Yaskawa INFORM job: OK_R2_O57-69(1)(90,0)_OK.JBI

/JOB
//NAME OK_R2_O57-69(1)(90,0)_OK
///FOLDERNAME X4
//POS
///NPOS 460,460,460,17,0,0
///TOOL 0
///POSTYPE PULSE
///PULSE
C00000=-107863,126513,61876,4074,92941,-4149
C00001=-107635,120046,52933,4022,95106,-4012
C00002=-107385,124787,62548,3925,91623,-4047
C00003=-107289,126429,66937,3891,89767,-4074
C00004=-107289,125685,67059,3890,89310,-4088
C00005=-107289,126429,66937,3891,89767,-4074
C00006=-107447,131976,74605,3936,87910,-4183
C00007=-107368,129085,70604,3913,88881,-4126
C00008=-107503,121805,59343,3962,92067,-4069
C00009=-107756,117289,50059,4061,95463,-4036
C00010=-108153,112100,52912,9904,92668,-10418
C00011=-107537,116907,62411,9707,89272,-10490
C00012=-107296,118643,67053,9639,87306,-10566
C00013=-107296,118210,67408,9641,86871,-10599
C00014=-107296,118643,67053,9639,87306,-10566
C00015=-106873,123308,73383,9530,85780,-10546
C00016=-107051,120523,69599,9574,86686,-10534
C00017=-107734,114067,59645,9761,89532,-10533
C00018=-108357,109439,50420,9963,92855,-10467
C00019=-111395,93808,29792,10909,97789,-10982
C00020=-122185,34205,35653,27729,49230,-19016
C00021=-120981,41909,45488,27980,46968,-19127
C00022=-117396,66636,64308,14609,59928,-14205
C00023=-117396,67398,66227,14722,59162,-14310
C00024=-117396,66924,65038,14651,59635,-14244
C00025=-117026,69424,68003,14605,59045,-14176
C00026=-117396,66924,65038,14651,59635,-14244
C00027=-121567,39659,44448,28509,46708,-19512
C00028=-122801,32028,34766,28268,48928,-19417
C00029=-122836,-30084,-33960,23424,71784,-41222
C00030=-108542,-18181,-29050,8736,76414,-35911
C00031=-108679,-18112,-25517,8852,74315,-36109
C00032=-108679,-17878,-23614,8896,73277,-36184
C00033=-108679,-18015,-24674,8871,73853,-36141
C00034=-101227,-12151,-22997,-5627,79968,-34149
C00035=-100809,-11793,-21323,-5732,79157,-33969
C00036=-99890,-11248,-20900,-5932,79243,-33658
C00037=-100809,-11793,-21323,-5732,79157,-33969
C00038=-119599,-28607,-38623,18108,79564,-38965
C00039=-143809,-13353,-27562,-4151,73883,-14363
C00040=-142866,3813,-3489,-4615,67955,-13814
C00041=-142866,4258,-993,-4658,66653,-13764
C00042=-142866,4067,-2013,-4640,67181,-13786
C00043=-143013,7668,1106,-4588,67106,-13835
C00044=-142866,4067,-2013,-4640,67181,-13786
C00045=-131729,19399,12333,-22118,77640,8494
C00046=-132684,19784,12695,-21959,77361,8191
C00047=-131729,18326,5882,-21907,80820,7904
C00048=-118180,-25123,-37779,-23861,88752,11312
C00049=-84402,-63677,-67114,-22586,99939,48241
C00050=-125926,-77250,-66316,-21080,81833,36437
C00051=-126284,-594,-20029,-15604,88354,35723
C00052=-126284,-509,-12976,-15645,84209,36248
C00053=-124802,3877,-7879,-15893,83645,36839
C00054=-124802,4020,-6552,-15911,82926,36931
C00055=-124802,3943,-7243,-15902,83298,36884
C00056=-123270,3785,-7378,-16131,83600,37383
C00057=-123399,3884,-6575,-16123,83149,37397
C00058=-123813,3922,-6544,-16060,83068,37263
C00059=-123399,3797,-7355,-16113,83568,37342
C00060=-129363,-46213,-49135,-15183,82438,35396
C00061=-131818,-93939,-91511,-4308,83147,7603
C00062=-129147,-104974,-80844,32439,31226,-48978
C00063=-125584,-72667,-62488,33742,33102,-67368
C00064=-122739,-67050,-57509,31022,31859,-65945
C00065=-121864,-64027,-53896,30654,30960,-65755
C00066=-121864,-63651,-52586,31182,30432,-66030
C00067=-121864,-64027,-53896,30654,30960,-65755
C00068=-121821,-59098,-51320,29827,31769,-65322
C00069=-121798,-56590,-49965,29444,32160,-65121
C00070=-121821,-59098,-51320,29827,31769,-65322
C00071=-130221,-55648,-47387,49393,39382,-72629
C00072=-128533,-55969,-47565,48393,38431,-72058
C00073=-122326,-63724,-54491,30711,31580,-65784
C00074=-123406,-65952,-56523,31749,32071,-66325
C00075=-126254,-71501,-61496,34397,33361,-67713
C00076=-120687,-90156,-48971,65843,10407,33929
C00077=-163424,-29173,-12092,69684,68620,47205
C00078=-167450,-15662,-2475,69350,71709,47134
C00079=-157670,-380,9649,68931,65290,48661
C00080=-176833,-62202,-56111,67907,81183,43629
C00081=-171503,-69579,-59831,67744,77015,43718
C00082=-167720,-72113,-59544,67781,73885,43604
C00083=-167720,-71727,-58313,67922,73661,43360
C00084=-167720,-72113,-59544,67781,73885,43604
C00085=-166558,-71597,-59299,67661,73156,43817
C00086=-165333,-70928,-58979,67520,72398,44056
C00087=-166558,-71597,-59299,67661,73156,43817
C00088=-171811,-70314,-60189,67797,77159,43607
C00089=-177694,-60868,-55413,67941,81861,43620
C00090=-178740,-64487,-57291,68086,82281,43176
C00091=-194893,-69888,-59984,68507,92693,40544
C00092=-214988,-85940,-67216,66402,104593,36100
C00093=-204042,-120915,-85873,62426,87530,23210
C00094=-200540,-66438,-67217,63628,100285,-15829
C00095=-127293,-88890,-117674,21964,112183,-47373
C00096=-127884,-113870,-117586,20406,100261,-49782
C00097=-126455,-94233,-83658,19548,96625,-49926
C00098=-122769,-95152,-80887,19686,93685,-49072
C00099=-121257,-92855,-76623,19731,91957,-48808
C00100=-121256,-92184,-75240,19721,91480,-48885
C00101=-121257,-92855,-76623,19731,91957,-48808
C00102=-119709,-92847,-76620,19813,91585,-48312
C00103=-118447,-92805,-76604,19874,91287,-47906
C00104=-121134,-93057,-78029,19757,92646,-48652
C00105=-122616,-92853,-79205,19699,93786,-49000
C00106=-126246,-91944,-81970,19569,96706,-49837
C00107=-116739,-91029,-87152,-11175,94833,69838
C00108=-118638,-93558,-84500,-11112,91693,69464
C00109=-121559,-94813,-81066,-11067,88585,68734
C00110=-121559,-94454,-79960,-11067,88097,68778
C00111=-121559,-94813,-81066,-11067,88585,68734
C00112=-121580,-97932,-82261,-11067,87731,68801
C00113=-121559,-94813,-81066,-11067,88585,68734
C00114=-124478,-94674,-81011,-11026,88221,67759
C00115=-121559,-94813,-81066,-11067,88585,68734
C00116=-121199,-93273,-83309,-11082,90766,68663
C00117=-119237,-90980,-86060,-11143,93854,69064
C00118=-119262,-91078,-98551,-11400,101347,68370
C00119=-119262,-88450,-105465,-11733,106843,67839
C00120=-123634,-129086,-124562,18007,62786,-21453
C00121=-124713,-112307,-109989,18584,62695,-21889
C00122=-121750,-102661,-104576,16897,63614,-20597
C00123=-120661,-96847,-100545,16291,63882,-20142
C00124=-120661,-96945,-99213,16408,63045,-20264
C00125=-120661,-96847,-100545,16291,63882,-20142
C00126=-119434,-96825,-100537,15680,63651,-19709
C00127=-118199,-96764,-100511,15059,63439,-19270
C00128=-119434,-96825,-100537,15680,63651,-19709
C00129=-120468,-95018,-99831,16130,64325,-20004
C00130=-120473,-92385,-98782,16042,65005,-19908
C00131=-120468,-95018,-99831,16130,64325,-20004
C00132=-121400,-102567,-103315,16828,62845,-20579
C00133=-124338,-112119,-108698,18515,61948,-21869
C00134=-115152,-110094,-108973,-21966,66789,27187
C00135=-118701,-101887,-103909,-20282,66922,25804
C00136=-120033,-96498,-99821,-19662,66842,25314
C00137=-120033,-96571,-98630,-19770,66116,25442
C00138=-120033,-96498,-99821,-19662,66842,25314
C00139=-121038,-96503,-99823,-19217,66607,24975
C00140=-122863,-96447,-99800,-18396,66209,24352
C00141=-121038,-96503,-99823,-19217,66607,24975
C00142=-121031,-93073,-98698,-19079,67622,24806
C00143=-121028,-91162,-97925,-19016,68103,24728
C00144=-121031,-93073,-98698,-19079,67622,24806
C00145=-119849,-101075,-102503,-19842,66224,25492
C00146=-116381,-109262,-107580,-21511,66068,26853
C00147=-114174,-113759,-109466,-25218,61256,29915
C00148=-117999,-105066,-104585,-23039,61495,28291
C00149=-119436,-99712,-100384,-22286,61259,27759
C00150=-119436,-99710,-99356,-22420,60673,27881
C00151=-119436,-99712,-100384,-22286,61259,27759
C00152=-121229,-99730,-100389,-21374,60785,27131
C00153=-123455,-99637,-100354,-20211,60254,26337
C00154=-121229,-99730,-100389,-21374,60785,27131
C00155=-121193,-87849,-97584,-20616,64895,26352
C00156=-121184,-85182,-96456,-20515,65531,26236
C00157=-121193,-87849,-97584,-20616,64895,26352
C00158=-119818,-94456,-100985,-21520,64018,27049
C00159=-116346,-102514,-105912,-23431,63914,28430
C00160=-120616,-96535,-104175,-23887,64719,45568
C00161=-120616,-96992,-102054,-24182,63306,45881
C00162=-136549,-91664,-102215,-2850,64532,40154
C00163=-118869,-97062,-101163,-25162,63282,46587
C00164=-120614,-98220,-102778,-24220,63138,45920
C00165=-133771,-94843,-111628,-11760,91195,37379
C00166=-135495,-95953,-105009,-10406,87462,38794
C00167=-135817,-95923,-103691,-10152,86855,39072
C00168=-120616,-96793,-103087,-23408,87451,42960
C00169=-120617,-96070,-105685,-23410,89266,42604
C00170=-120635,-118119,-124325,-17957,114364,37370
C00171=-107148,-122068,-106720,-37591,45003,56343
C00172=-107143,-118125,-97071,-40168,41922,57944
C00173=-107140,-117153,-94914,-40772,41285,58308
C00174=-108761,-111076,-92035,-38763,41593,57087
C00175=-105115,-116142,-93852,-42098,42144,59139
C00176=-107012,-118507,-95796,-40965,41228,58425
C00177=-106625,-124982,-112623,-27698,77800,49761
C00178=-108670,-124346,-112001,-25564,83023,48254
C00179=-122914,-112386,-108022,-9565,118901,48106
C00180=-107149,-124464,-114807,-14035,115464,42498
C00181=-107153,-124980,-118069,-14274,117155,42276
C00182=-120683,-72727,-118704,-1403,106780,1205
C00183=-120616,-97084,-101761,23685,56760,-46645
C00184=-120615,-97341,-97713,24403,54354,-47226
C00185=-120615,-97245,-95574,24781,53197,-47519
C00186=-113473,-96585,-93861,15515,48754,-41599
C00187=-120613,-98403,-96349,24817,53089,-47545
C00188=-122362,-97151,-94697,25998,53280,-48291
C00189=-118726,-95773,-106258,22948,89010,-41713
C00190=-118527,-107245,-109313,22939,85243,-42364
C00191=-120617,-95328,-107797,23350,90604,-42068
C00192=-120618,-93989,-110172,23402,92584,-41681
C00193=-120619,-87370,-116055,23793,99045,-40394
C00194=-120619,-87370,-116055,23793,99045,-40394
C00195=-120618,-86394,-114990,-8935,74593,-77376
C00196=-120618,-89943,-112390,-9089,71210,-77123
C00197=-120618,-91094,-111253,-9157,69935,-77026
C00198=-120921,-87010,-110025,-8929,71231,-77225
C00199=-120616,-91696,-112687,-9127,70502,-77069
C00200=-120617,-91433,-110915,-9280,69085,-76949
C00201=-120617,-91707,-110620,-9342,68290,-76888
C00202=-120617,-92092,-110153,-9289,66860,-76810
C00203=-120617,-92703,-109346,-8604,64312,-76688
C00204=-120617,-93084,-108807,-7222,62458,-76641
C00205=-120617,-93193,-108666,-5837,61715,-76664
C00206=-120618,-90875,-111661,-5103,64613,-76670
C00207=-120618,-90809,-111742,-4197,64653,-76687
C00208=-120618,-90545,-112027,-2634,65244,-76730
C00209=-120618,-90001,-112556,-1051,66686,-76779
C00210=-120618,-89211,-113241,130,68806,-76818
C00211=-120618,-88484,-113805,667,70701,-76840
C00212=-120618,-87123,-114601,725,72803,-76709
C00213=-120619,-86169,-115177,666,75079,-76754
C00214=-120619,-85009,-115798,-44,77805,-76866
C00215=-120619,-84186,-116189,-1368,79788,-77043
C00216=-120619,-83945,-116287,-2643,80551,-77203
C00217=-118270,-87908,-113898,-4548,77310,-76315
C00218=-117006,-87882,-113777,-5977,77383,-75992
C00219=-115001,-87936,-113393,-8376,77055,-75464
C00220=-113157,-88199,-112730,-10795,75966,-74930
C00221=-112003,-88721,-111920,-12625,74164,-74513
C00222=-111959,-89151,-111512,-13141,72976,-74431
C00223=-114352,-90005,-111461,-12180,71784,-75105
C00224=-117604,-90791,-111341,-10710,70486,-76060
C00225=-117404,-89600,-112462,-10735,71791,-76111
C00226=-116906,-85938,-115017,-10812,75246,-76259
C00227=-120614,-97623,-100799,-20300,88883,51757
C00228=-120614,-96302,-87355,-20440,81742,52958
C00229=-120613,-95405,-83784,-20521,80111,53236
C00230=-127344,-108772,-84900,-17713,65232,40253
C00231=-119108,-93712,-82042,-20736,80300,53753
C00232=-120703,-96440,-84059,-20528,79748,53266
C00233=-121654,-94959,-82200,-16195,85067,56749
C00234=-121447,-94482,-79045,-16244,83477,57034
C00235=-120534,-97306,-80078,-13287,88870,68293
C00236=-120613,-95181,-82964,-13310,91650,67966
C00237=-120614,-96223,-86939,-13345,93512,67766
C00238=-120615,-97634,-95801,-13498,98116,67263
C00239=-121294,-114205,-91205,24827,58618,-34956
C00240=-120612,-94063,-79189,30374,49118,-27390
C00241=-120612,-92317,-74276,31337,47279,-28045
C00242=-120611,-91635,-72532,31685,46659,-28276
C00243=-117825,-85297,-69483,27706,45876,-25590
C00244=-120609,-92794,-73597,31655,46709,-28256
C00245=-122365,-91337,-71823,32796,47086,-29053
C00246=-115287,-110447,-90354,20374,67075,-37718
C00247=-116232,-100454,-77072,21254,66209,-40580
C00248=-116013,-94136,-76050,20295,81458,-56297
C00249=-120612,-93792,-78416,23522,88402,-60481
C00250=-120613,-94966,-82014,23532,89885,-60189
C00251=-192979,-49879,-84133,31949,90821,-59300
C00252=-226136,-49296,-77583,43048,96139,-60221
C00253=-194231,-43574,-37464,64429,96533,35524
C00254=-168190,-921,2356,69742,86936,65420
C00255=-167171,-9679,-4727,69794,80481,66551
C00256=-161668,-12899,-4972,71887,72051,48991
C00257=-157343,-12771,-6150,68681,68498,39910
C00258=-156881,-17849,-10944,69825,79076,66625
C00259=-156054,-17027,-11609,69675,78824,67093
C00260=-157320,-12846,-6207,68680,68481,39912
C00261=-155303,-14498,-7398,68413,65801,40416
C00262=-150761,-18705,-10675,67104,57790,42164
C00263=-154138,4950,8277,69166,76187,38481
C00264=-154445,-11009,-7055,66235,75211,55885
C00265=-154064,-10379,-10377,61252,81435,65690
C00266=-159305,-13086,-7363,68622,70046,39902
C00267=-160610,-11568,-6196,68690,70948,39749
C00268=-179726,-19719,-12316,69264,83687,37039
C00269=-180202,-65513,-36112,70171,79517,38597
C00270=-171321,-47804,-23743,70196,73038,45095
C00271=-120855,-117042,-83065,287,50429,-281
C00272=-120852,-56541,-79529,233,79340,-219
C00273=-120696,51333,26745,175,69370,-180
C00274=-120686,107911,74673,172,68949,-177
C00275=-120685,95088,60632,169,71000,-174
C00276=-122318,97205,64688,817,69601,-751
C00277=-120685,108202,77433,173,67399,-179
C00278=-120704,104217,73450,180,67803,-185
C00279=-122286,97202,64700,804,69591,-740
C00280=-121454,98107,65862,475,69334,-448
C00281=-120585,97922,65623,2034,69446,-1841
C00282=-122017,99369,67601,7878,69886,-7136
C00283=-124401,105713,75936,15606,71119,-14640
C00284=-128119,115493,91326,26372,70058,-18277
C00285=-128088,115464,91288,26362,70055,-18265
C00286=-119886,111402,95174,38234,57086,-30403
C00287=-120666,108818,81293,29360,75518,-26461
C00288=-140740,108253,75800,14319,69459,-12393
C00289=-141155,96820,62941,14306,71509,-12294
C00290=-143909,115216,86261,19079,74712,-18279
C00291=-140740,108512,78347,14450,68068,-12565
C00292=-141173,105757,75971,14609,68190,-12710
C00293=-142377,104065,71962,18453,77277,-17320
C00294=-143915,117471,89727,22794,77825,-23537
C00295=-139477,109798,84410,35996,86879,-36501
C00296=-140751,108928,81956,36051,87607,-36108
C00297=-140752,108346,78971,36051,88864,-35697
C00298=-147823,62894,38016,27898,90947,-27507
C00299=-160213,20954,5847,52912,104038,-48859
C00300=-159152,20729,17995,59071,100827,-50067
C00301=-155802,40777,37843,59069,97737,-50212
C00302=-160195,38796,31307,59203,102054,-49818
C00303=-156773,55935,3033,15469,106475,-467
C00304=-153918,39963,-12238,-14336,97152,19223
C00305=-159942,42906,-84,-7000,88493,12017
C00306=-161832,44450,4966,-4658,85344,9495
C00307=-160451,43537,6688,-5079,83896,9996
C00308=-170176,47751,11203,12092,85800,-8664
C00309=-172574,61876,26837,20283,90605,-20342
C00310=-175474,59660,23243,20803,92313,-21058
C00311=-176824,52719,4578,21456,100048,-20156
C00312=-152577,48148,-11201,-5231,110173,9097
C00313=-182779,-40861,-76585,4205,87735,83212
C00314=-189334,-126614,-108463,44477,62316,64668
C00315=-120096,-126434,-88762,51835,16555,74218
C00316=-139248,-82584,-73342,59042,45862,69599
C00317=-136350,-83647,-73803,58003,43942,70198
C00318=-130421,-76673,-73912,46604,46265,76427
C00319=-135820,-86240,-74234,58721,43036,69743
C00320=-135177,-84196,-74622,57263,43352,70634
C00321=-130462,-76664,-73908,46626,46288,76415
C00322=-118284,-90424,-77484,27464,26422,76602
C00323=-134750,-71454,-68054,46452,38063,58888
C00324=-143711,-58767,-60463,57749,51756,38253
C00325=-120675,-86248,-74914,23863,24288,53303
C00326=-120674,-86256,-74917,23863,24286,53303
C00327=-120096,-126434,-88762,51835,16555,74218
C00328=-118534,-85327,-101542,-31688,82312,3081
C00329=-123235,4833,-40404,-29868,88268,-211
C00330=-160796,40344,30640,-17217,54638,-7315
C00331=-160797,40341,30637,-17217,54638,-7315
C00332=-160797,40341,30637,-17217,54638,-7315
C00333=-160252,39151,28676,-17378,55324,-7200
C00334=-161178,38223,28434,-16963,54814,-7508
C00335=-160796,40350,30646,-17218,54637,-7315
C00336=-160795,40351,30648,-17218,54637,-7314
C00337=-160794,40354,30651,-17218,54637,-7314
C00338=-134054,6396,-12292,-27269,70214,305
C00339=-134055,6392,-12295,-27269,70214,305
C00340=-134055,6392,-12295,-27269,70214,305
C00341=-133335,6117,-13247,-27465,70843,432
C00342=-134208,4264,-14132,-27207,70198,248
C00343=-134055,6400,-12288,-27269,70214,305
C00344=-134054,6402,-12286,-27269,70214,305
C00345=-134054,6405,-12283,-27270,70214,305
C00346=-134054,6378,-12307,-27269,70215,305
C00347=-110297,97127,46558,-158,86609,-5885
C00348=-106536,103923,39499,6534,95353,-6477
C00349=-105914,112602,52325,6316,91893,-6465
C00350=-107411,115180,62232,6738,87264,-7175
C00351=-107307,119116,66280,6709,86790,-7167
C00352=-105927,112591,52310,6320,91897,-6469
C00353=-107439,122836,73336,-765,83341,-3278
C00354=-107821,123137,73841,-645,83181,-3398
C00355=-102914,145277,103073,-11065,82212,10729
C00356=-102506,149279,108574,-13236,82700,14235
C00357=-102941,142782,99507,-15695,87156,18184
C00358=-102438,125149,73506,-15865,93942,17486
C00359=-103348,95167,36366,-12069,90690,17205
C00360=-107306,118463,66661,-801,85196,-3245
C00361=-107311,128667,66498,14067,94509,-10827
C00362=-105409,128969,69208,9127,93984,-11176
C00363=-104752,117595,57274,7632,88999,-11570
C00364=-107310,126688,66629,14039,93443,-10948
C00365=-107566,122823,62593,14116,93966,-10970
C00366=-105955,108102,46748,11418,87672,-11524
C00367=-106075,110081,48628,12407,89224,-11272
C00368=-104774,107445,45071,11972,89867,-10810
C00369=-104167,107349,44943,11766,89817,-10628
C00370=-103614,108174,46048,11576,89495,-10489
C00371=-105019,105279,39955,12261,92654,-10576
C00372=-107312,128730,66586,14067,94488,-10830
C00373=-113054,107191,42951,15619,98894,-12042
C00374=-132655,20555,-34602,20500,105579,-17250
C00375=-120395,-75677,-109491,17431,99945,-14261
C00376=-120731,-81008,-115648,-105,86416,-81801
C00377=-120675,-24654,-47163,-132,73228,-81771
C00378=-120676,-24640,-47153,-131,73229,-81771
C00379=-121102,-22780,-44290,48,72423,-81914
C00380=-120676,-24370,-48215,-131,74021,-81772
C00381=-121750,-24626,-47144,317,73232,-82133
C00382=-121088,-18910,-41523,41,72708,-81911
C00383=-120676,-24640,-47153,-131,73229,-81771
C00384=-120672,-32524,-49889,-133,70864,-81769
C00385=-86683,-40445,-63075,-13763,77736,-70672
C00386=-103499,26970,-9106,-7161,77072,-76192
C00387=-140778,108078,66600,-20509,92089,-48724
C00388=-140778,108101,66629,-20508,92083,-48723
C00389=-140777,108123,66659,-20508,92077,-48722
C00390=-140791,110557,71328,-20474,90549,-48468
C00391=-140777,108420,65802,-20527,92715,-48830
C00392=-141368,109052,67884,-20414,91674,-48860
C00393=-140538,117676,80864,-20492,88534,-48038
C00394=-140777,108123,66659,-20508,92077,-48722
C00395=-140778,108101,66629,-20508,92083,-48723
C00396=-140778,108101,66629,-20508,92083,-48723
C00397=-140778,108122,66658,-20508,92077,-48722
C00398=-140768,108703,68758,-20489,91145,-48562
C00399=-140777,108420,65801,-20527,92715,-48830
C00400=-141368,109051,67883,-20414,91674,-48860
C00401=-140511,115176,77354,-20500,89363,-48171
C00402=-140778,108122,66658,-20508,92077,-48722
C00403=-140778,108100,66628,-20508,92083,-48723
C00404=-140778,108078,66599,-20509,92089,-48724
C00405=-126581,14025,-47477,-25241,115824,-48542
C00406=-159492,92702,46653,-29136,105568,-44545
C00407=-162149,88036,41181,-28914,105145,-45798
C00408=-163325,88052,47564,-28312,101300,-45262
C00409=-160866,111719,71725,-28335,100123,-43674
C00410=-160864,108336,66000,-28535,101703,-44070
C00411=-164354,88224,47874,-28236,100875,-45547
C00412=-160866,108108,66623,-28476,101259,-43959
C00413=-161429,110004,69125,-28389,100573,-44000
C00414=-160867,107600,68720,-43807,97992,-44930
C00415=-160869,107245,72152,-43546,96305,-44200
C00416=-160853,112270,81548,-43267,93953,-43186
C00417=-160872,111361,79145,-43345,94689,-43509
C00418=-160869,107230,72446,-43527,96165,-44140
C00419=-161852,112523,81931,-43214,93388,-43402
C00420=-160870,107231,72133,-43547,96307,-44201
C00421=-160868,107586,68702,-43807,97995,-44932
C00422=-160873,107541,68625,-43810,98010,-44941
C00423=-160875,107181,72050,-43549,96324,-44211
C00424=-160969,112164,81513,-43259,93871,-43205
C00425=-160878,111286,79028,-43348,94711,-43521
C00426=-160875,107165,72344,-43530,96184,-44151
C00427=-161946,112277,81723,-43208,93342,-43426
C00428=-160876,107167,72031,-43549,96326,-44212
C00429=-160874,107528,68607,-43810,98012,-44942
C00430=-160865,108116,66633,-19225,80466,79641
C00431=-160864,108012,67019,-19239,80191,79685
C00432=-160902,111102,73963,-19378,77641,80084
C00433=-160868,111461,73140,-19346,78303,79987
C00434=-160865,107941,67240,-19247,80028,79711
C00435=-161896,111383,74336,-19093,77331,79779
C00436=-160866,107998,67001,-19238,80195,79684
C00437=-160866,108102,66615,-19224,80470,79640
C00438=-141960,25007,-13534,-18907,77065,75548
C00439=-148396,38776,-224,-4331,80270,75408
C00440=-147937,42862,4060,-4507,79758,75574
C00441=-147586,38479,-2882,-4613,81790,75612
C00442=-132676,28155,-16568,-22865,92034,69453
C00443=-139622,-24488,-52979,-20482,85647,66084
C00444=-105595,-117820,-100492,-25848,75539,72989
C00445=-106580,-108863,-97500,-25415,77736,72126
C00446=-109054,-118504,-91401,-16987,64899,66879
C00447=-114351,-116427,-87550,-15194,62531,65147
C00448=-119485,-94955,-76898,-12502,65960,62737
C00449=-99170,-109633,-81201,-29999,68590,70531
C00450=-97263,-108225,-79726,-30318,69111,71170
C00451=-119688,-71486,-66798,-11989,71648,62069
C00452=-119489,-72073,-70371,-11931,73536,61952
C00453=-119715,-43131,-54580,-11630,78554,61387
C00454=-119934,-43288,-51446,-11646,76556,61502
C00455=-120006,-17553,-34071,-11532,79027,61243
C00456=-119832,-16968,-37707,-11506,81540,61066
C00457=-138269,-21321,-44343,15851,46320,74175
C00458=-176671,-154466,-104215,64912,39697,45563
C00459=-34524,-124554,-102946,40349,70974,61921
BC00000=290556,778984,53
BC00001=296477,827832,53
BC00002=296477,827832,53
BC00003=296477,827832,52
BC00004=296477,827832,52
BC00005=296477,827832,52
BC00006=296477,827832,52
BC00007=296477,827832,52
BC00008=296477,827832,53
BC00009=296477,827832,53
BC00010=305680,824697,66927
BC00011=305680,824697,66927
BC00012=305680,824697,66927
BC00013=305680,824697,66927
BC00014=305680,824697,66927
BC00015=305680,824697,66927
BC00016=305680,824697,66927
BC00017=305680,824697,66927
BC00018=305680,824697,66927
BC00019=305680,824697,66927
BC00020=269068,808420,256770
BC00021=269068,808420,256770
BC00022=269068,808420,256770
BC00023=269068,808420,256770
BC00024=269068,808420,256770
BC00025=269068,808420,256770
BC00026=269068,808420,256770
BC00027=269068,808420,256770
BC00028=269068,808420,256770
BC00029=269068,808420,256770
BC00030=269068,808420,256770
BC00031=269068,808420,256770
BC00032=269068,808420,256770
BC00033=269068,808420,256770
BC00034=269068,808420,256770
BC00035=269068,808420,256770
BC00036=269068,808420,256770
BC00037=269068,808420,256770
BC00038=269068,808420,256770
BC00039=269068,808420,256770
BC00040=269068,808420,256770
BC00041=269068,808420,256770
BC00042=269068,808420,256770
BC00043=269068,808420,256770
BC00044=269068,808420,256770
BC00045=269068,808420,256770
BC00046=269068,808420,256770
BC00047=269068,808420,256770
BC00048=269068,808420,256770
BC00049=269068,722620,256770
BC00050=178494,722620,256770
BC00051=178494,722620,256770
BC00052=178494,722620,256770
BC00053=178494,722620,256770
BC00054=178494,722620,256770
BC00055=178494,722620,256770
BC00056=178494,722620,256770
BC00057=178494,722620,256770
BC00058=178494,722620,256770
BC00059=178494,722620,256770
BC00060=178494,722620,256770
BC00061=138756,709064,202273
BC00062=61964,682869,96959
BC00063=15,683519,90542
BC00064=15,683519,90542
BC00065=15,683519,90542
BC00066=15,683519,90542
BC00067=15,683519,90542
BC00068=15,683519,90542
BC00069=15,683519,90542
BC00070=15,683519,90542
BC00071=15,683519,90542
BC00072=15,683519,90542
BC00073=15,683519,90542
BC00074=15,683519,90542
BC00075=15,683519,90542
BC00076=1273,683756,232707
BC00077=15,671225,229408
BC00078=15,671225,229408
BC00079=16,671226,229406
BC00080=15,740766,97992
BC00081=15,744979,78990
BC00082=15,746665,71384
BC00083=15,746665,71384
BC00084=15,746665,71384
BC00085=15,746665,71384
BC00086=15,746665,71384
BC00087=15,746665,71384
BC00088=15,744091,71514
BC00089=15,739878,90515
BC00090=15,739878,90515
BC00091=15,739878,90515
BC00092=15,739878,90515
BC00093=4537,733723,217212
BC00094=80822,696048,563603
BC00095=35157,680076,1075175
BC00096=35157,770360,1075175
BC00097=34361,771324,1075175
BC00098=34361,771324,1075175
BC00099=34361,771324,1075175
BC00100=34361,771324,1075175
BC00101=34361,771324,1075175
BC00102=34361,771324,1075175
BC00103=34361,771324,1075175
BC00104=34361,771324,1075175
BC00105=34361,771324,1075175
BC00106=34361,771324,1075175
BC00107=42797,766692,1075175
BC00108=42797,766692,1075175
BC00109=42797,766692,1075175
BC00110=42797,766692,1075175
BC00111=42797,766692,1075175
BC00112=42797,766692,1075175
BC00113=42797,766692,1075175
BC00114=42797,766692,1075175
BC00115=42797,766692,1075175
BC00116=42797,766692,1075175
BC00117=42797,766692,1075175
BC00118=42797,766692,1075175
BC00119=42797,766692,1075175
BC00120=146022,859779,1075175
BC00121=146022,859779,1075175
BC00122=146022,859779,1075175
BC00123=146022,859779,1075175
BC00124=146022,859779,1075175
BC00125=146022,859779,1075175
BC00126=146022,859779,1075175
BC00127=146022,859779,1075175
BC00128=146022,859779,1075175
BC00129=146022,859779,1075175
BC00130=146022,859779,1075175
BC00131=146022,859779,1075175
BC00132=146022,859779,1075175
BC00133=146022,859779,1075175
BC00134=176049,857561,1075175
BC00135=176049,857561,1075175
BC00136=176049,857561,1075175
BC00137=176049,857561,1075175
BC00138=176049,857561,1075175
BC00139=176049,857561,1075175
BC00140=176049,857561,1075175
BC00141=176049,857561,1075175
BC00142=176049,857561,1075175
BC00143=176049,857561,1075175
BC00144=176049,857561,1075175
BC00145=176049,857561,1075175
BC00146=176049,857561,1075175
BC00147=129734,841826,1075175
BC00148=129734,841826,1075175
BC00149=129734,841826,1075175
BC00150=129734,841826,1075175
BC00151=129734,841826,1075175
BC00152=129734,841826,1075175
BC00153=129734,841826,1075175
BC00154=129734,841826,1075175
BC00155=129734,841826,1075175
BC00156=129734,841826,1075175
BC00157=129734,841826,1075175
BC00158=129734,841826,1075175
BC00159=129734,841826,1075175
BC00160=142153,845657,1075175
BC00161=136701,849303,1075175
BC00162=134520,850762,1075175
BC00163=134520,850762,1075175
BC00164=134520,850762,1075175
BC00165=137516,886222,1075172
BC00166=137720,849041,1075174
BC00167=137762,841415,1075175
BC00168=140007,840932,1075175
BC00169=145619,839727,1075175
BC00170=180456,929432,1075175
BC00171=168021,846183,1075175
BC00172=168042,846186,1075175
BC00173=163006,851102,1075175
BC00174=160992,853068,1075175
BC00175=160992,853068,1075175
BC00176=160992,853068,1075175
BC00177=169557,896858,1075175
BC00178=171239,895275,1075172
BC00179=158426,945505,1075171
BC00180=160107,947347,1075175
BC00181=164973,949360,1075175
BC00182=157894,860706,1075175
BC00183=127221,848277,1075175
BC00184=127232,848278,1075175
BC00185=132508,852516,1075175
BC00186=134618,854212,1075171
BC00187=134619,854211,1075175
BC00188=134619,854211,1075175
BC00189=128708,899486,1075175
BC00190=128708,899486,1075175
BC00191=126448,894646,1075175
BC00192=120840,893399,1075175
BC00193=120819,893396,1075175
BC00194=108659,806260,1075175
BC00195=397033,866889,1075175
BC00196=396343,869401,1075175
BC00197=396067,870405,1075175
BC00198=396067,870405,1075175
BC00199=396067,870405,1075175
BC00200=391503,868887,1075175
BC00201=388851,867701,1075175
BC00202=387842,866199,1075175
BC00203=385581,863689,1075175
BC00204=382314,862051,1075175
BC00205=379450,861705,1075175
BC00206=374365,881250,1075175
BC00207=372628,881564,1075175
BC00208=369853,882526,1075175
BC00209=367245,884287,1075175
BC00210=365527,886651,1075175
BC00211=365120,888691,1075175
BC00212=386897,893714,1075175
BC00213=387767,895993,1075175
BC00214=389889,898568,1075175
BC00215=393093,900280,1075175
BC00216=395952,900656,1075175
BC00217=398174,881178,1075175
BC00218=398174,880854,1075175
BC00219=398174,879840,1075175
BC00220=398174,877989,1075175
BC00221=398174,875535,1075175
BC00222=398174,874097,1075175
BC00223=398174,872876,1075175
BC00224=398174,871457,1075175
BC00225=398174,870453,1075175
BC00226=398174,867941,1075175
BC00227=52330,766929,1075175
BC00228=52330,766929,1075175
BC00229=47260,766939,1075175
BC00230=45232,766943,1075175
BC00231=45232,766943,1075175
BC00232=45232,766943,1075175
BC00233=39669,775379,1075175
BC00234=48611,761121,1075175
BC00235=43094,771298,1075175
BC00236=44336,772357,1075175
BC00237=47441,775005,1075175
BC00238=47420,775002,1075175
BC00239=32781,783617,1075175
BC00240=26171,746916,1075175
BC00241=26181,746918,1075175
BC00242=30773,752599,1075175
BC00243=32609,754871,1075175
BC00244=32609,754871,1075175
BC00245=32609,754871,1075175
BC00246=29513,796201,1075175
BC00247=29656,745498,1075175
BC00248=30736,758476,1075175
BC00249=29625,769411,1075175
BC00250=24737,771387,1075175
BC00251=181441,722385,1075175
BC00252=206367,695978,993979
BC00253=43511,699656,343050
BC00254=15,700638,169199
BC00255=15,700493,176682
BC00256=15,702608,172046
BC00257=15,703868,169284
BC00258=15,702762,156281
BC00259=15,702762,156281
BC00260=15,703868,169284
BC00261=15,698813,169275
BC00262=15,689550,169221
BC00263=15,686170,169200
BC00264=15,699513,166456
BC00265=15,707199,164860
BC00266=15,702130,176769
BC00267=15,697786,195480
BC00268=15,697786,195480
BC00269=15,703831,213681
BC00270=15,696835,229408
BC00271=302372,698952,211490
BC00272=302372,717858,201268
BC00273=302372,750216,183774
BC00274=305532,747625,53
BC00275=305569,761849,53
BC00276=305584,765283,53
BC00277=305584,756031,53
BC00278=305584,756031,53
BC00279=305584,765283,53
BC00280=305584,765283,53
BC00281=305584,765283,53
BC00282=305584,765283,53
BC00283=305584,765283,53
BC00284=305584,765283,53
BC00285=305584,765283,53
BC00286=242092,730480,4
BC00287=254268,725168,543
BC00288=373423,757548,53
BC00289=374646,771594,53
BC00290=375136,780484,53
BC00291=375136,766039,53
BC00292=375136,766039,53
BC00293=375136,780484,53
BC00294=375136,780484,53
BC00295=326830,797507,51
BC00296=324367,796451,53
BC00297=318212,793809,53
BC00298=331956,796432,138844
BC00299=331956,796432,138844
BC00300=331956,796432,138844
BC00301=331956,796432,138844
BC00302=331956,796432,138844
BC00303=345139,769043,66616
BC00304=345139,804305,66616
BC00305=345139,804305,66616
BC00306=345139,804305,66616
BC00307=345139,804305,66616
BC00308=345139,804305,66616
BC00309=345139,804305,66616
BC00310=345139,804305,66616
BC00311=345139,804305,66616
BC00312=349847,779193,40824
BC00313=390673,737123,107565
BC00314=230273,714746,68332
BC00315=15,702747,12011
BC00316=15,701955,18543
BC00317=15,706339,2244
BC00318=15,708068,108
BC00319=15,708093,53
BC00320=15,708093,53
BC00321=15,708068,108
BC00322=15,708068,108
BC00323=13937,696226,53
BC00324=526,700184,53
BC00325=47,698020,1277
BC00326=766,691948,17562
BC00327=15,702747,12011
BC00328=297950,700262,124402
BC00329=297950,699644,21134
BC00330=369493,695491,225137
BC00331=365725,700831,210595
BC00332=364218,702968,204778
BC00333=364218,702968,204778
BC00334=364218,702968,204778
BC00335=366008,702976,196139
BC00336=367515,700839,201956
BC00337=371283,695499,216499
BC00338=284979,736274,157916
BC00339=281211,741614,143374
BC00340=279704,743751,137557
BC00341=279704,743751,137557
BC00342=279704,743751,137557
BC00343=281466,743758,129052
BC00344=282973,741622,134869
BC00345=286741,736281,149411
BC00346=286720,736279,203179
BC00347=296348,799025,115750
BC00348=298529,835561,48149
BC00349=299550,837400,19199
BC00350=299550,828814,63772
BC00351=299550,828814,63772
BC00352=299550,837400,19199
BC00353=302497,828021,63552
BC00354=297997,829570,63542
BC00355=297997,829570,63542
BC00356=297997,829570,63542
BC00357=297997,829570,63542
BC00358=297997,829570,63542
BC00359=297979,829494,63811
BC00360=296254,822118,90028
BC00361=285994,828831,497
BC00362=289766,832894,53
BC00363=289766,832895,51
BC00364=291275,834519,53
BC00365=291275,834519,53
BC00366=293188,832323,52
BC00367=301226,828160,53
BC00368=301226,828160,53
BC00369=301226,828160,53
BC00370=301226,828160,53
BC00371=301517,827668,53
BC00372=299924,819919,440
BC00373=301049,820896,39095
BC00374=304889,824233,171046
BC00375=304889,700105,171046
BC00376=83775,699365,9536
BC00377=83778,689858,175427
BC00378=83769,691199,148957
BC00379=83766,691735,138369
BC00380=83766,691735,138369
BC00381=83766,691735,138369
BC00382=83766,691735,138369
BC00383=83757,694806,148969
BC00384=83766,693464,175440
BC00385=83763,737347,138110
BC00386=83763,737347,138110
BC00387=197029,737142,72736
BC00388=197039,737143,45852
BC00389=197033,737820,19073
BC00390=197030,738091,8361
BC00391=197030,738091,8361
BC00392=197030,738091,8361
BC00393=197030,738091,8361
BC00394=197021,741431,19085
BC00395=197027,740754,45864
BC00396=196907,776675,45988
BC00397=196900,777352,19209
BC00398=196894,778679,8502
BC00399=196898,777623,8498
BC00400=196898,777623,8498
BC00401=196894,778679,8502
BC00402=196889,780936,19222
BC00403=196895,780259,46001
BC00404=196885,780258,72885
BC00405=171385,775077,62173
BC00406=212214,724112,35449
BC00407=211106,741301,33281
BC00408=211106,741301,33281
BC00409=211368,723652,53
BC00410=211368,723652,53
BC00411=211106,741301,33281
BC00412=208356,721958,8668
BC00413=223868,722216,29649
BC00414=206229,720775,53
BC00415=203870,719461,53
BC00416=202410,718648,52
BC00417=202926,718936,53
BC00418=202926,718936,53
BC00419=202410,718648,52
BC00420=200593,717623,53
BC00421=202951,718937,53
BC00422=191785,744837,53
BC00423=189426,743524,53
BC00424=188187,742833,51
BC00425=188482,742998,53
BC00426=188482,742998,53
BC00427=188187,742833,51
BC00428=186209,741719,53
BC00429=188567,743033,53
BC00430=212591,717178,21939
BC00431=210233,715864,53
BC00432=209289,715339,53
BC00433=209289,715339,53
BC00434=209289,715339,53
BC00435=209289,715339,53
BC00436=206956,714026,53
BC00437=209314,715340,21939
BC00438=192907,721782,82797
BC00439=192907,721782,82797
BC00440=192907,721782,82797
BC00441=192907,721782,82797
BC00442=184359,725138,114504
BC00443=179787,742375,125459
BC00444=167642,738874,171871
BC00445=167642,765336,159298
BC00446=157612,789455,186175
BC00447=157612,789455,186175
BC00448=157612,789455,186175
BC00449=157612,789455,186175
BC00450=157612,789455,186175
BC00451=157612,789455,186175
BC00452=157612,789455,186175
BC00453=157612,789455,186175
BC00454=157612,789455,186175
BC00455=157612,789455,186175
BC00456=157612,789455,186175
BC00457=164113,763380,121188
BC00458=164113,711732,121188
BC00459=279725,698376,1053175
EC00000=798156,0
EC00001=798156,0
EC00002=798156,0
EC00003=798156,0
EC00004=798156,0
EC00005=798156,0
EC00006=798156,0
EC00007=798156,0
EC00008=798156,0
EC00009=798156,0
EC00010=798156,0
EC00011=798156,0
EC00012=798156,0
EC00013=798156,0
EC00014=798156,0
EC00015=798156,0
EC00016=798156,0
EC00017=798156,0
EC00018=798156,0
EC00019=798156,0
EC00020=798156,0
EC00021=798156,0
EC00022=798156,0
EC00023=798156,0
EC00024=798156,0
EC00025=798156,0
EC00026=798156,0
EC00027=798156,0
EC00028=798156,0
EC00029=798156,0
EC00030=798156,0
EC00031=798156,0
EC00032=798156,0
EC00033=798156,0
EC00034=798156,0
EC00035=798156,0
EC00036=798156,0
EC00037=798156,0
EC00038=798156,0
EC00039=798156,0
EC00040=798156,0
EC00041=798156,0
EC00042=798156,0
EC00043=798156,0
EC00044=798156,0
EC00045=798156,0
EC00046=798156,0
EC00047=798156,0
EC00048=798156,0
EC00049=798156,0
EC00050=798156,0
EC00051=798156,0
EC00052=798156,0
EC00053=798156,0
EC00054=798156,0
EC00055=798156,0
EC00056=798156,0
EC00057=798156,0
EC00058=798156,0
EC00059=798156,0
EC00060=798156,0
EC00061=798156,0
EC00062=798156,0
EC00063=798156,0
EC00064=798156,0
EC00065=798156,0
EC00066=798156,0
EC00067=798156,0
EC00068=798156,0
EC00069=798156,0
EC00070=798156,0
EC00071=798156,0
EC00072=798156,0
EC00073=798156,0
EC00074=798156,0
EC00075=798156,0
EC00076=798156,0
EC00077=798156,0
EC00078=798156,0
EC00079=798154,0
EC00080=798156,0
EC00081=798156,0
EC00082=798156,0
EC00083=798156,0
EC00084=798156,0
EC00085=798156,0
EC00086=798156,0
EC00087=798156,0
EC00088=798156,0
EC00089=798156,0
EC00090=798156,0
EC00091=798156,0
EC00092=798156,0
EC00093=820978,0
EC00094=883374,0
EC00095=975524,0
EC00096=975524,0
EC00097=975524,0
EC00098=975524,0
EC00099=975524,0
EC00100=975524,0
EC00101=975524,0
EC00102=975524,0
EC00103=975524,0
EC00104=975524,0
EC00105=975524,0
EC00106=975524,0
EC00107=975524,0
EC00108=975524,0
EC00109=975524,0
EC00110=975524,0
EC00111=975524,0
EC00112=975524,0
EC00113=975524,0
EC00114=975524,0
EC00115=975524,0
EC00116=975524,0
EC00117=975524,0
EC00118=975524,0
EC00119=975524,0
EC00120=975524,0
EC00121=975524,0
EC00122=975524,0
EC00123=975524,0
EC00124=975524,0
EC00125=975524,0
EC00126=975524,0
EC00127=975524,0
EC00128=975524,0
EC00129=975524,0
EC00130=975524,0
EC00131=975524,0
EC00132=975524,0
EC00133=975524,0
EC00134=975524,0
EC00135=975524,0
EC00136=975524,0
EC00137=975524,0
EC00138=975524,0
EC00139=975524,0
EC00140=975524,0
EC00141=975524,0
EC00142=975524,0
EC00143=975524,0
EC00144=975524,0
EC00145=975524,0
EC00146=975524,0
EC00147=975524,0
EC00148=975524,0
EC00149=975524,0
EC00150=975524,0
EC00151=975524,0
EC00152=975524,0
EC00153=975524,0
EC00154=975524,0
EC00155=975524,0
EC00156=975524,0
EC00157=975524,0
EC00158=975524,0
EC00159=975524,0
EC00160=975524,0
EC00161=975524,0
EC00162=975524,0
EC00163=975524,0
EC00164=975524,0
EC00165=975521,1
EC00166=975523,0
EC00167=975524,0
EC00168=975524,0
EC00169=975524,0
EC00170=975524,0
EC00171=975524,0
EC00172=975524,0
EC00173=975524,0
EC00174=975524,0
EC00175=975524,0
EC00176=975524,0
EC00177=975524,0
EC00178=975521,1
EC00179=975522,0
EC00180=975524,0
EC00181=975524,0
EC00182=975524,0
EC00183=975524,0
EC00184=975524,0
EC00185=975524,0
EC00186=975521,0
EC00187=975524,0
EC00188=975524,0
EC00189=975524,0
EC00190=975524,0
EC00191=975524,0
EC00192=975524,0
EC00193=975524,0
EC00194=975524,0
EC00195=975524,0
EC00196=975524,0
EC00197=975524,0
EC00198=975524,0
EC00199=975524,0
EC00200=975524,0
EC00201=975524,0
EC00202=975524,0
EC00203=975524,0
EC00204=975524,0
EC00205=975524,0
EC00206=975524,0
EC00207=975524,0
EC00208=975524,0
EC00209=975524,0
EC00210=975524,0
EC00211=975524,0
EC00212=975524,0
EC00213=975524,0
EC00214=975524,0
EC00215=975524,0
EC00216=975524,0
EC00217=975524,0
EC00218=975524,0
EC00219=975524,0
EC00220=975524,0
EC00221=975524,0
EC00222=975524,0
EC00223=975524,0
EC00224=975524,0
EC00225=975524,0
EC00226=975524,0
EC00227=975524,0
EC00228=975524,0
EC00229=975524,0
EC00230=975524,0
EC00231=975524,0
EC00232=975524,0
EC00233=975524,0
EC00234=975524,0
EC00235=975524,0
EC00236=975524,0
EC00237=975524,0
EC00238=975524,0
EC00239=975524,0
EC00240=975524,0
EC00241=975524,0
EC00242=975524,0
EC00243=975524,0
EC00244=975524,0
EC00245=975524,0
EC00246=975524,0
EC00247=975524,0
EC00248=975524,0
EC00249=975524,0
EC00250=975524,0
EC00251=975524,0
EC00252=959628,0
EC00253=832192,0
EC00254=798156,0
EC00255=798156,0
EC00256=798156,0
EC00257=798156,0
EC00258=798156,0
EC00259=798156,0
EC00260=798156,0
EC00261=798156,0
EC00262=798156,0
EC00263=798156,0
EC00264=798156,0
EC00265=798156,0
EC00266=798156,0
EC00267=798156,0
EC00268=798156,0
EC00269=798156,0
EC00270=798156,0
EC00271=798156,0
EC00272=798156,0
EC00273=798156,0
EC00274=798156,0
EC00275=798156,0
EC00276=798156,0
EC00277=798156,0
EC00278=798156,0
EC00279=798156,0
EC00280=798156,0
EC00281=798156,0
EC00282=798156,0
EC00283=798156,0
EC00284=798156,0
EC00285=798156,0
EC00286=798156,0
EC00287=798156,0
EC00288=798156,0
EC00289=798156,0
EC00290=798156,0
EC00291=798156,0
EC00292=798156,0
EC00293=798156,0
EC00294=798156,0
EC00295=798154,1
EC00296=798156,0
EC00297=798156,0
EC00298=798156,0
EC00299=798156,0
EC00300=798156,0
EC00301=798156,0
EC00302=798156,0
EC00303=798156,0
EC00304=798156,0
EC00305=798156,0
EC00306=798156,0
EC00307=798156,0
EC00308=798156,0
EC00309=798156,0
EC00310=798156,0
EC00311=798156,0
EC00312=798156,0
EC00313=798156,0
EC00314=798156,0
EC00315=798156,0
EC00316=798156,0
EC00317=798156,0
EC00318=798156,0
EC00319=798156,0
EC00320=798156,0
EC00321=798156,0
EC00322=798156,0
EC00323=798156,0
EC00324=798156,0
EC00325=798156,0
EC00326=798156,0
EC00327=798156,0
EC00328=798156,0
EC00329=798156,0
EC00330=798156,0
EC00331=798156,0
EC00332=798156,0
EC00333=798156,0
EC00334=798156,0
EC00335=798156,0
EC00336=798156,0
EC00337=798156,0
EC00338=798156,0
EC00339=798156,0
EC00340=798156,0
EC00341=798156,0
EC00342=798156,0
EC00343=798156,0
EC00344=798156,0
EC00345=798156,0
EC00346=798156,0
EC00347=798156,0
EC00348=798156,0
EC00349=798156,0
EC00350=798156,0
EC00351=798156,0
EC00352=798156,0
EC00353=798156,0
EC00354=798155,1
EC00355=798155,1
EC00356=798155,1
EC00357=798155,1
EC00358=798155,1
EC00359=798155,1
EC00360=798156,0
EC00361=798156,0
EC00362=798156,0
EC00363=798155,0
EC00364=798156,0
EC00365=798156,0
EC00366=798156,0
EC00367=798156,0
EC00368=798156,0
EC00369=798156,0
EC00370=798156,0
EC00371=798156,0
EC00372=798156,0
EC00373=798156,0
EC00374=798156,0
EC00375=798156,0
EC00376=798156,0
EC00377=798156,0
EC00378=798156,0
EC00379=798156,0
EC00380=798156,0
EC00381=798156,0
EC00382=798156,0
EC00383=798156,0
EC00384=798156,0
EC00385=798156,0
EC00386=798156,0
EC00387=798156,0
EC00388=798156,0
EC00389=798156,0
EC00390=798156,0
EC00391=798156,0
EC00392=798156,0
EC00393=798156,0
EC00394=798156,0
EC00395=798156,0
EC00396=798156,0
EC00397=798156,0
EC00398=798156,0
EC00399=798156,0
EC00400=798156,0
EC00401=798156,0
EC00402=798156,0
EC00403=798156,0
EC00404=798156,0
EC00405=798156,0
EC00406=798156,0
EC00407=798156,0
EC00408=798156,0
EC00409=798156,0
EC00410=798156,0
EC00411=798156,0
EC00412=798156,0
EC00413=798156,0
EC00414=798156,0
EC00415=798156,0
EC00416=798155,0
EC00417=798156,0
EC00418=798156,0
EC00419=798155,0
EC00420=798156,0
EC00421=798156,0
EC00422=798156,0
EC00423=798156,0
EC00424=798154,1
EC00425=798156,0
EC00426=798156,0
EC00427=798154,1
EC00428=798156,0
EC00429=798156,0
EC00430=798156,0
EC00431=798156,0
EC00432=798156,0
EC00433=798156,0
EC00434=798156,0
EC00435=798156,0
EC00436=798156,0
EC00437=798156,0
EC00438=798156,0
EC00439=798156,0
EC00440=798156,0
EC00441=798156,0
EC00442=798156,0
EC00443=798156,0
EC00444=798156,0
EC00445=798156,0
EC00446=798156,0
EC00447=798156,0
EC00448=798156,0
EC00449=798156,0
EC00450=798156,0
EC00451=798156,0
EC00452=798156,0
EC00453=798156,0
EC00454=798156,0
EC00455=798156,0
EC00456=798156,0
EC00457=798156,0
EC00458=798156,0
EC00459=798156,0
///POSTYPE BASE
///RECTAN
///RCONF 0,0,0,0,0,0,0,0,0,0,0,0,0,0,0,0,0,0,0,0,0,0,0,0
P00006=0.222,-3.123,-1.508,0.0000,0.0000,0.0000
P00021=-0.225,-6.128,-0.405,0.0000,0.0000,0.0000
P00022=0.222,-3.123,-1.508,0.0000,0.0000,0.0000
P00024=0.145,-0.552,1.326,0.0000,0.0000,0.0000
P00025=-2.003,0.006,0.728,0.0000,0.0000,0.0000
P00026=0.562,-0.002,-0.337,0.0000,0.0000,0.0000
P00027=-0.746,0.015,-9.096,0.0000,0.0000,0.0000
P00032=1.957,0.503,-7.217,0.0000,0.0000,0.0000
P00041=0.192,3.924,0.305,0.0000,0.0000,0.0000
P00042=-0.217,1.941,0.413,0.0000,0.0000,0.0000
P00043=-0.044,-1.937,1.197,0.0000,0.0000,0.0000
P00044=0.687,-2.322,1.156,0.0000,0.0000,0.0000
P00045=-0.068,-0.810,1.603,0.0000,0.0000,0.0000
P00046=0.799,0.043,1.292,0.0000,0.0000,0.0000
P00066=5.557,-0.028,3.115,0.0000,0.0000,0.0000
///RCONF 0,1,0,0,0,0,0,0,0,0,0,0,0,0,0,0,0,0,0,0,0,0,0,0
P00067=-0.081,0.026,-1.119,0.0000,0.0000,0.0000
///RCONF 0,0,0,0,0,0,0,0,0,0,0,0,0,0,0,0,0,0,0,0,0,0,0,0
P00068=2.896,1.192,4.622,0.0000,0.0000,0.0000
//INST
///DATE 2025/02/07 12:48
///ATTR SC,RW
///GROUP1 RB1,BS1
///GROUP2 ST1
NOP
'OK_r2_O57-69(1)(90,0)
'Down
'Path S1900
SFTOF3D
'Path S1901
SFTOF3D
MOVJ C00000 BC00000 VJ=40.00  +MOVJ EC00000 VJ=15.00
MOVJ C00001 BC00001 VJ=100.00  +MOVJ EC00001 VJ=100.00
MOVL C00002 BC00002 V=400.0  +MOVJ EC00002 VJ=100.00
SMOVL C00003 BC00003 V=100.0  +MOVJ EC00003
SREFP 3 C00004 BC00004  +REFP EC00004
CALL JOB:SEARCH-R1-S13D
SET P026 P006
SFTON3D P026
SMOVL C00005 BC00005 V=100.0  +MOVJ EC00005
SREFP 3 C00006 BC00006  +REFP EC00006
CALL JOB:SEARCH-R1-S13D
SET P026 P006
SFTON3D P026
SMOVL C00007 BC00007 V=100.0  +MOVJ EC00007
MOVL C00008 BC00008 V=400.0  +MOVJ EC00008 VJ=100.00
MOVL C00009 BC00009 V=1000.0  +MOVJ EC00009 VJ=100.00
'Path S1902
SFTOF3D
MOVJ C00010 BC00010 VJ=100.00  +MOVJ EC00010 VJ=100.00
MOVL C00011 BC00011 V=400.0  +MOVJ EC00011 VJ=100.00
SMOVL C00012 BC00012 V=100.0  +MOVJ EC00012
SREFP 3 C00013 BC00013  +REFP EC00013
CALL JOB:SEARCH-R1-S13D
SET P027 P006
SFTON3D P027
SMOVL C00014 BC00014 V=100.0  +MOVJ EC00014
SREFP 3 C00015 BC00015  +REFP EC00015
CALL JOB:SEARCH-R1-S13D
SET P027 P006
SFTON3D P027
SMOVL C00016 BC00016 V=100.0  +MOVJ EC00016
SFTOF3D
MOVL C00017 BC00017 V=400.0  +MOVJ EC00017 VJ=100.00
MOVL C00018 BC00018 V=1000.0  +MOVJ EC00018 VJ=100.00
MOVJ C00019 BC00019 VJ=100.00  +MOVJ EC00019 VJ=100.00
'Path S1903
SFTOF3D
MOVJ C00020 BC00020 VJ=100.00  +MOVJ EC00020 VJ=100.00
COMM PAUSE
COMM MOVL C00021 BC00021 V=400.0  +MOVJ EC00021 VJ=100.00
COMM SMOVL C00022 BC00022 V=100.0  +MOVJ EC00022
COMM SREFP 3 C00023 BC00023  +REFP EC00023
COMM CALL JOB:SEARCH-R1-S13D
COMM SET P022 P006
COMM SFTON3D P022
COMM SMOVL C00024 BC00024 V=100.0  +MOVJ EC00024
COMM SREFP 3 C00025 BC00025  +REFP EC00025
COMM CALL JOB:SEARCH-R1-S13D
COMM SET P022 P006
COMM SFTON3D P022
COMM SMOVL C00026 BC00026 V=100.0  +MOVJ EC00026
COMM SFTOF3D
COMM MOVL C00027 BC00027 V=400.0  +MOVJ EC00027 VJ=100.00
COMM MOVL C00028 BC00028 V=1000.0  +MOVJ EC00028 VJ=100.00
SMOVL C00029 BC00029 V=1000.0  +MOVJ EC00029
SMOVL C00030 BC00030 V=1000.0  +MOVJ EC00030
SMOVL C00031 BC00031 V=166.7  +MOVJ EC00031
SREFP 3 C00032 BC00032  +REFP EC00032
CALL JOB:SEARCH-R1-S13D
SET P066 P006
SFTON3D P066
SMOVL C00033 BC00033 V=250.0  +MOVJ EC00033
SMOVL C00034 BC00034 V=250.0  +MOVJ EC00034
SMOVL C00035 BC00035 V=250.0  +MOVJ EC00035
SREFP 3 C00036 BC00036  +REFP EC00036
CALL JOB:SEARCH-R1-S13D
SET P066 P006
SFTON3D P066
SMOVL C00037 BC00037 V=250.0  +MOVJ EC00037
SMOVL C00038 BC00038 V=1000.0  +MOVJ EC00038
SFTOF3D
SMOVL C00039 BC00039 V=1000.0  +MOVJ EC00039
SMOVL C00040 BC00040 V=166.7  +MOVJ EC00040
SREFP 3 C00041 BC00041  +REFP EC00041
CALL JOB:SEARCH-R1-S13D
SET P068 P006
SFTON3D P068
SMOVL C00042 BC00042 V=250.0  +MOVJ EC00042
SREFP 3 C00043 BC00043  +REFP EC00043
CALL JOB:SEARCH-R1-S13D
SET P068 P006
SFTON3D P068
SMOVL C00044 BC00044 V=250.0  +MOVJ EC00044
SMOVL C00045 BC00045 V=166.7  +MOVJ EC00045
SREFP 3 C00046 BC00046  +REFP EC00046
CALL JOB:SEARCH-R1-S13D
SET P068 P006
SFTON3D P068
SMOVL C00047 BC00047 V=250.0  +MOVJ EC00047
SFTOF3D
SMOVL C00048 BC00048 V=1000.0  +MOVJ EC00048
MOVJ C00049 BC00049 VJ=100.00  +MOVJ EC00049 VJ=100.00
MOVJ C00050 BC00050 VJ=100.00  +MOVJ EC00050 VJ=100.00
COMM PAUSE
COMM MOVJ C00051 BC00051 VJ=100.00  +MOVJ EC00051 VJ=100.00
COMM SMOVL C00052 BC00052 V=1000.0  +MOVJ EC00052
COMM SMOVL C00053 BC00053 V=166.7  +MOVJ EC00053
COMM SREFP 3 C00054 BC00054  +REFP EC00054
COMM CALL JOB:SEARCH-R1-S13D
COMM SET P067 P006
COMM SFTON3D P067
COMM SMOVL C00055 BC00055 V=250.0  +MOVJ EC00055
COMM SMOVL C00056 BC00056 V=250.0  +MOVJ EC00056
COMM SMOVL C00057 BC00057 V=133.3  +MOVJ EC00057
COMM SREFP 3 C00058 BC00058  +REFP EC00058
COMM CALL JOB:SEARCH-R1-S13D
COMM SET P067 P006
COMM SFTON3D P067
COMM SMOVL C00059 BC00059 V=250.0  +MOVJ EC00059
COMM SFTOF3D
COMM SMOVL C00060 BC00060 V=1000.0  +MOVJ EC00060
SMOVL C00061 BC00061 V=1000.0  +MOVJ EC00061
MOVJ C00062 BC00062 VJ=100.00  +MOVJ EC00062 VJ=50.00
MOVJ C00063 BC00063 VJ=100.00  +MOVJ EC00063 VJ=100.00
MOVL C00064 BC00064 V=400.0  +MOVJ EC00064 VJ=100.00
SMOVL C00065 BC00065 V=100.0  +MOVJ EC00065
SREFP 3 C00066 BC00066  +REFP EC00066
CALL JOB:SEARCH-R1-S13D
SET P021 P006
SFTON3D P021
SMOVL C00067 BC00067 V=100.0  +MOVJ EC00067
SMOVL C00068 BC00068 V=100.0  +MOVJ EC00068
SREFP 3 C00069 BC00069  +REFP EC00069
CALL JOB:SEARCH-R1-S13D
SET P021 P006
SFTON3D P021
SMOVL C00070 BC00070 V=100.0  +MOVJ EC00070
SMOVL C00071 BC00071 V=100.0  +MOVJ EC00071
SREFP 3 C00072 BC00072  +REFP EC00072
CALL JOB:SEARCH-R1-S13D
SET P021 P006
SFTON3D P021
SMOVL C00073 BC00073 V=100.0  +MOVJ EC00073
MOVL C00074 BC00074 V=400.0  +MOVJ EC00074 VJ=100.00
MOVL C00075 BC00075 V=1000.0  +MOVJ EC00075 VJ=100.00
MOVJ C00076 BC00076 VJ=100.00  +MOVJ EC00076 VJ=100.00
MOVJ C00077 BC00077 VJ=100.00  +MOVJ EC00077 VJ=100.00
MOVJ C00078 BC00078 VJ=100.00  +MOVJ EC00078 VJ=100.00
MOVJ C00079 BC00079 VJ=100.00  +MOVJ EC00079 VJ=100.00
'Path S1912
SFTOF3D
MOVJ C00080 BC00080 VJ=100.00  +MOVJ EC00080 VJ=100.00
MOVL C00081 BC00081 V=400.0  +MOVJ EC00081 VJ=100.00
SMOVL C00082 BC00082 V=100.0  +MOVJ EC00082
SREFP 3 C00083 BC00083  +REFP EC00083
CALL JOB:SEARCH-R1-S13D
SET P032 P006
SFTON3D P032
SMOVL C00084 BC00084 V=100.0  +MOVJ EC00084
SMOVL C00085 BC00085 V=100.0  +MOVJ EC00085
SREFP 3 C00086 BC00086  +REFP EC00086
CALL JOB:SEARCH-R1-S13D
SET P032 P006
SFTON3D P032
SMOVL C00087 BC00087 V=100.0  +MOVJ EC00087
SFTOF3D
MOVL C00088 BC00088 V=400.0  +MOVJ EC00088 VJ=100.00
MOVL C00089 BC00089 V=1000.0  +MOVJ EC00089 VJ=100.00
MOVJ C00090 BC00090 VJ=100.00  +MOVJ EC00090 VJ=100.00
MOVJ C00091 BC00091 VJ=100.00  +MOVJ EC00091 VJ=100.00
'Up
MOVJ C00092 BC00092 VJ=100.00  +MOVJ EC00092 VJ=50.00
MOVJ C00093 BC00093 VJ=100.00  +MOVJ EC00093 VJ=100.00
MOVJ C00094 BC00094 VJ=100.00  +MOVJ EC00094 VJ=100.00
MOVJ C00095 BC00095 VJ=100.00  +MOVJ EC00095 VJ=100.00
MOVJ C00096 BC00096 VJ=100.00  +MOVJ EC00096 VJ=100.00
'Path S1137
SFTOF3D
MOVJ C00097 BC00097 VJ=100.00  +MOVJ EC00097 VJ=100.00
MOVL C00098 BC00098 V=400.0  +MOVJ EC00098 VJ=100.00
SMOVL C00099 BC00099 V=100.0  +MOVJ EC00099
SREFP 3 C00100 BC00100  +REFP EC00100
CALL JOB:SEARCH-R1-S13D
SET P046 P006
SFTON3D P046
SMOVL C00101 BC00101 V=100.0  +MOVJ EC00101
SMOVL C00102 BC00102 V=100.0  +MOVJ EC00102
SREFP 3 C00103 BC00103  +REFP EC00103
CALL JOB:SEARCH-R1-S13D
SET P046 P006
SFTON3D P046
SMOVL C00104 BC00104 V=100.0  +MOVJ EC00104
MOVL C00105 BC00105 V=400.0  +MOVJ EC00105 VJ=100.00
MOVL C00106 BC00106 V=1000.0  +MOVJ EC00106 VJ=100.00
'Path S1169
SFTOF3D
MOVJ C00107 BC00107 VJ=100.00  +MOVJ EC00107 VJ=100.00
MOVL C00108 BC00108 V=400.0  +MOVJ EC00108 VJ=100.00
SMOVL C00109 BC00109 V=100.0  +MOVJ EC00109
SREFP 3 C00110 BC00110  +REFP EC00110
CALL JOB:SEARCH-R1-S13D
SET P045 P006
SFTON3D P045
SMOVL C00111 BC00111 V=100.0  +MOVJ EC00111
SREFP 3 C00112 BC00112  +REFP EC00112
CALL JOB:SEARCH-R1-S13D
SET P045 P006
SFTON3D P045
SMOVL C00113 BC00113 V=100.0  +MOVJ EC00113
SREFP 3 C00114 BC00114  +REFP EC00114
CALL JOB:SEARCH-R1-S13D
SET P045 P006
SFTON3D P045
SMOVL C00115 BC00115 V=100.0  +MOVJ EC00115
SFTOF3D
MOVL C00116 BC00116 V=400.0  +MOVJ EC00116 VJ=100.00
MOVL C00117 BC00117 V=1000.0  +MOVJ EC00117 VJ=100.00
MOVL C00118 BC00118 V=1000.0  +MOVJ EC00118 VJ=100.00
MOVJ C00119 BC00119 VJ=100.00  +MOVJ EC00119 VJ=50.00
MOVJ C00120 BC00120 VJ=100.00  +MOVJ EC00120 VJ=50.00
MOVJ C00121 BC00121 VJ=100.00  +MOVJ EC00121 VJ=100.00
MOVL C00122 BC00122 V=400.0  +MOVJ EC00122 VJ=100.00
SMOVL C00123 BC00123 V=100.0  +MOVJ EC00123
SREFP 3 C00124 BC00124  +REFP EC00124
CALL JOB:SEARCH-R1-S13D
SET P043 P006
SFTON3D P043
SMOVL C00125 BC00125 V=100.0  +MOVJ EC00125
SMOVL C00126 BC00126 V=100.0  +MOVJ EC00126
SREFP 3 C00127 BC00127  +REFP EC00127
CALL JOB:SEARCH-R1-S13D
SET P043 P006
SFTON3D P043
SMOVL C00128 BC00128 V=100.0  +MOVJ EC00128
SMOVL C00129 BC00129 V=100.0  +MOVJ EC00129
SREFP 3 C00130 BC00130  +REFP EC00130
CALL JOB:SEARCH-R1-S13D
SET P043 P006
SFTON3D P043
SMOVL C00131 BC00131 V=100.0  +MOVJ EC00131
MOVL C00132 BC00132 V=400.0  +MOVJ EC00132 VJ=100.00
MOVL C00133 BC00133 V=1000.0  +MOVJ EC00133 VJ=100.00
'Path S1166
SFTOF3D
MOVJ C00134 BC00134 VJ=100.00  +MOVJ EC00134 VJ=100.00
MOVL C00135 BC00135 V=400.0  +MOVJ EC00135 VJ=100.00
SMOVL C00136 BC00136 V=100.0  +MOVJ EC00136
SREFP 3 C00137 BC00137  +REFP EC00137
CALL JOB:SEARCH-R1-S13D
SET P042 P006
SFTON3D P042
SMOVL C00138 BC00138 V=100.0  +MOVJ EC00138
SMOVL C00139 BC00139 V=100.0  +MOVJ EC00139
SREFP 3 C00140 BC00140  +REFP EC00140
CALL JOB:SEARCH-R1-S13D
SET P042 P006
SFTON3D P042
SMOVL C00141 BC00141 V=100.0  +MOVJ EC00141
SMOVL C00142 BC00142 V=100.0  +MOVJ EC00142
SREFP 3 C00143 BC00143  +REFP EC00143
CALL JOB:SEARCH-R1-S13D
SET P042 P006
SFTON3D P042
SMOVL C00144 BC00144 V=100.0  +MOVJ EC00144
MOVL C00145 BC00145 V=400.0  +MOVJ EC00145 VJ=100.00
MOVL C00146 BC00146 V=1000.0  +MOVJ EC00146 VJ=100.00
'Path S1165
SFTOF3D
MOVJ C00147 BC00147 VJ=100.00  +MOVJ EC00147 VJ=100.00
MOVL C00148 BC00148 V=400.0  +MOVJ EC00148 VJ=100.00
SMOVL C00149 BC00149 V=100.0  +MOVJ EC00149
SREFP 3 C00150 BC00150  +REFP EC00150
CALL JOB:SEARCH-R1-S13D
SET P041 P006
SFTON3D P041
SMOVL C00151 BC00151 V=100.0  +MOVJ EC00151
SMOVL C00152 BC00152 V=100.0  +MOVJ EC00152
SREFP 3 C00153 BC00153  +REFP EC00153
CALL JOB:SEARCH-R1-S13D
SET P041 P006
SFTON3D P041
SMOVL C00154 BC00154 V=100.0  +MOVJ EC00154
SMOVL C00155 BC00155 V=100.0  +MOVJ EC00155
SREFP 3 C00156 BC00156  +REFP EC00156
CALL JOB:SEARCH-R1-S13D
SET P041 P006
SFTON3D P041
SMOVL C00157 BC00157 V=100.0  +MOVJ EC00157
MOVL C00158 BC00158 V=400.0  +MOVJ EC00158 VJ=100.00
MOVL C00159 BC00159 V=1000.0  +MOVJ EC00159 VJ=100.00
'Path W378
SFTOF3D
SFTON3D P041
MOVJ C00160 BC00160 VJ=100.00  +MOVJ EC00160 VJ=100.00
SMOVL C00161 BC00161 V=400.0  +MOVJ EC00161
SMOVL C00162 BC00162 V=133.3 PL=0  +MOVJ EC00162
SREFP 1 C00163 BC00163  +REFP EC00163
SREFP 2 C00164 BC00164  +REFP EC00164
MACRO1 MJ#(0) ARGF9
ARCON
SWVON WEV#(61)
SMOVL C00165 BC00165 V=6.7  +MOVJ EC00165
SMOVL C00166 BC00166 V=6.7  +MOVJ EC00166
SMOVL C00167 BC00167 V=6.7  +MOVJ EC00167
ARCOF
SWVOF
SMOVL C00168 BC00168 V=400.0  +MOVJ EC00168
SMOVL C00169 BC00169 V=1000.0  +MOVJ EC00169
SFTOF3D
MOVJ C00170 BC00170 VJ=100.00  +MOVJ EC00170 VJ=100.00
'Path W379
SFTOF3D
SFTON3D P042
MOVJ C00171 BC00171 VJ=100.00  +MOVJ EC00171 VJ=100.00
MOVJ C00172 BC00172 VJ=100.00  +MOVJ EC00172 VJ=100.00
SMOVL C00173 BC00173 V=400.0  +MOVJ EC00173
SMOVL C00174 BC00174 V=133.3 PL=0  +MOVJ EC00174
SREFP 1 C00175 BC00175  +REFP EC00175
SREFP 2 C00176 BC00176  +REFP EC00176
MACRO1 MJ#(0) ARGF9
ARCON
SMOVL C00177 BC00177 V=9.2  +MOVJ EC00177
SMOVL C00178 BC00178 V=9.2  +MOVJ EC00178
SMOVL C00179 BC00179 V=9.2  +MOVJ EC00179
ARCOF
SMOVL C00180 BC00180 V=400.0  +MOVJ EC00180
SMOVL C00181 BC00181 V=1000.0  +MOVJ EC00181
SFTOF3D
MOVJ C00182 BC00182 VJ=20.00  +MOVJ EC00182 VJ=100.00
'Path W380
SFTOF3D
SFTON3D P043
MOVJ C00183 BC00183 VJ=100.00  +MOVJ EC00183 VJ=100.00
MOVJ C00184 BC00184 VJ=100.00  +MOVJ EC00184 VJ=100.00
SMOVL C00185 BC00185 V=400.0  +MOVJ EC00185
SMOVL C00186 BC00186 V=133.3 PL=0  +MOVJ EC00186
SREFP 1 C00187 BC00187  +REFP EC00187
SREFP 2 C00188 BC00188  +REFP EC00188
ARCON
SMOVL C00189 BC00189 V=9.2  +MOVJ EC00189
SMOVL C00190 BC00190 V=9.2  +MOVJ EC00190
ARCOF
SMOVL C00191 BC00191 V=400.0  +MOVJ EC00191
SMOVL C00192 BC00192 V=1000.0  +MOVJ EC00192
SMOVL C00193 BC00193 V=1000.0  +MOVJ EC00193
MOVJ C00194 BC00194 VJ=100.00  +MOVJ EC00194 VJ=100.00
SFTOF3D
'NIE SPAWAMY
COMM 'Path W381
COMM SFTOF3D
COMM SFTON3D P044
COMM MOVJ C00195 BC00195 VJ=100.00  +MOVJ EC00195 VJ=100.00
COMM SMOVL C00196 BC00196 V=400.0  +MOVJ EC00196
COMM SMOVL C00197 BC00197 V=100.0 PL=0  +MOVJ EC00197
COMM SREFP 1 C00198 BC00198  +REFP EC00198
COMM SREFP 2 C00199 BC00199  +REFP EC00199
COMM MACRO1 MJ#(0) ARGF0
COMM ARCON
COMM SMOVL C00200 BC00200 V=10.0  +MOVJ EC00200
COMM SMOVL C00201 BC00201 V=10.0  +MOVJ EC00201
COMM SMOVL C00202 BC00202 V=10.0  +MOVJ EC00202
COMM SMOVL C00203 BC00203 V=10.0  +MOVJ EC00203
COMM SMOVL C00204 BC00204 V=10.0  +MOVJ EC00204
COMM SMOVL C00205 BC00205 V=10.0  +MOVJ EC00205
COMM SMOVL C00206 BC00206 V=10.0  +MOVJ EC00206
COMM SMOVL C00207 BC00207 V=10.0  +MOVJ EC00207
COMM SMOVL C00208 BC00208 V=10.0  +MOVJ EC00208
COMM SMOVL C00209 BC00209 V=10.0  +MOVJ EC00209
COMM SMOVL C00210 BC00210 V=10.0  +MOVJ EC00210
COMM SMOVL C00211 BC00211 V=10.0  +MOVJ EC00211
COMM SMOVL C00212 BC00212 V=10.0  +MOVJ EC00212
COMM SMOVL C00213 BC00213 V=10.0  +MOVJ EC00213
COMM SMOVL C00214 BC00214 V=10.0  +MOVJ EC00214
COMM SMOVL C00215 BC00215 V=10.0  +MOVJ EC00215
COMM SMOVL C00216 BC00216 V=10.0  +MOVJ EC00216
COMM SMOVL C00217 BC00217 V=10.0  +MOVJ EC00217
COMM SMOVL C00218 BC00218 V=10.0  +MOVJ EC00218
COMM SMOVL C00219 BC00219 V=10.0  +MOVJ EC00219
COMM SMOVL C00220 BC00220 V=10.0  +MOVJ EC00220
COMM SMOVL C00221 BC00221 V=10.0  +MOVJ EC00221
COMM SMOVL C00222 BC00222 V=10.0  +MOVJ EC00222
COMM SMOVL C00223 BC00223 V=10.0  +MOVJ EC00223
COMM SMOVL C00224 BC00224 V=10.0  +MOVJ EC00224
COMM ARCOF
COMM SMOVL C00225 BC00225 V=400.0  +MOVJ EC00225
COMM SMOVL C00226 BC00226 V=1000.0  +MOVJ EC00226
COMM SFTOF3D
'Path W382
SFTOF3D
MOVJ C00227 BC00227 VJ=100.00  +MOVJ EC00227 VJ=50.00
SFTON3D P045
MOVJ C00228 BC00228 VJ=100.00  +MOVJ EC00228 VJ=100.00
SMOVL C00229 BC00229 V=400.0  +MOVJ EC00229
SMOVL C00230 BC00230 V=133.3 PL=0  +MOVJ EC00230
SREFP 1 C00231 BC00231  +REFP EC00231
SREFP 2 C00232 BC00232  +REFP EC00232
ARCON
SMOVL C00233 BC00233 V=9.2  +MOVJ EC00233
SMOVL C00234 BC00234 V=9.2  +MOVJ EC00234
SMOVL C00235 BC00235 V=9.2  +MOVJ EC00235
ARCOF
SMOVL C00236 BC00236 V=400.0  +MOVJ EC00236
SMOVL C00237 BC00237 V=1000.0  +MOVJ EC00237
SMOVL C00238 BC00238 V=1000.0  +MOVJ EC00238
SFTOF3D
MOVJ C00239 BC00239 VJ=100.00  +MOVJ EC00239 VJ=100.00
'Path W383
SFTOF3D
SFTON3D P046
MOVJ C00240 BC00240 VJ=100.00  +MOVJ EC00240 VJ=100.00
MOVJ C00241 BC00241 VJ=100.00  +MOVJ EC00241 VJ=100.00
SMOVL C00242 BC00242 V=400.0  +MOVJ EC00242
SMOVL C00243 BC00243 V=133.3 PL=0  +MOVJ EC00243
SREFP 1 C00244 BC00244  +REFP EC00244
SREFP 2 C00245 BC00245  +REFP EC00245
ARCON
SMOVL C00246 BC00246 V=9.2  +MOVJ EC00246
SMOVL C00247 BC00247 V=9.2  +MOVJ EC00247
SMOVL C00248 BC00248 V=9.2  +MOVJ EC00248
ARCOF
SMOVL C00249 BC00249 V=400.0  +MOVJ EC00249
SMOVL C00250 BC00250 V=1000.0  +MOVJ EC00250
SFTOF3D
MOVJ C00251 BC00251 VJ=100.00  +MOVJ EC00251 VJ=100.00
MOVJ C00252 BC00252 VJ=100.00  +MOVJ EC00252 VJ=100.00
'Down
MOVJ C00253 BC00253 VJ=100.00  +MOVJ EC00253 VJ=100.00
MOVJ C00254 BC00254 VJ=100.00  +MOVJ EC00254 VJ=100.00
'Path W1720
SFTOF3D
SFTON3D P032
MOVJ C00255 BC00255 VJ=100.00  +MOVJ EC00255 VJ=100.00
SMOVL C00256 BC00256 V=400.0  +MOVJ EC00256
SMOVL C00257 BC00257 V=133.3  +MOVJ EC00257
SREFP 1 C00258 BC00258  +REFP EC00258
SREFP 2 C00259 BC00259  +REFP EC00259
MACRO1 MJ#(0) ARGF21
ARCON
SWVON WEV#(100)
SMOVC C00260 BC00260 V=9.2  +MOVJ EC00260
SMOVC C00261 BC00261 V=9.2  +MOVJ EC00261
SMOVC C00262 BC00262 V=9.2  +MOVJ EC00262
SMOVC C00263 BC00263 V=9.2  +MOVJ EC00263
SMOVC C00264 BC00264 V=9.2  +MOVJ EC00264
SMOVC C00265 BC00265 V=9.2  +MOVJ EC00265
ARCOF
SWVOF
SMOVL C00266 BC00266 V=400.0  +MOVJ EC00266
SMOVL C00267 BC00267 V=1000.0  +MOVJ EC00267
SFTOF3D
MOVJ C00268 BC00268 VJ=100.00  +MOVJ EC00268 VJ=100.00
MOVJ C00269 BC00269 VJ=100.00  +MOVJ EC00269 VJ=100.00
MOVJ C00270 BC00270 VJ=100.00  +MOVJ EC00270 VJ=100.00
MOVJ C00271 BC00271 VJ=100.00  +MOVJ EC00271 VJ=100.00
MOVJ C00272 BC00272 VJ=100.00  +MOVJ EC00272 VJ=100.00
MOVJ C00273 BC00273 VJ=100.00  +MOVJ EC00273 VJ=100.00
'Path W1626
SFTOF3D
COMM PAUSE
COMM SFTON3D P022
COMM MOVJ C00274 BC00274 VJ=100.00  +MOVJ EC00274 VJ=100.00
COMM SMOVL C00275 BC00275 V=250.0  +MOVJ EC00275
COMM SMOVL C00276 BC00276 V=133.3 PL=0  +MOVJ EC00276
COMM SREFP 1 C00277 BC00277  +REFP EC00277
COMM SREFP 2 C00278 BC00278  +REFP EC00278
COMM MACRO1 MJ#(0) ARGF9
COMM ARCON
COMM SMOVC C00279 BC00279 V=9.2  +MOVJ EC00279
COMM SMOVC C00280 BC00280 V=10.0  +MOVJ EC00280
COMM SMOVC C00281 BC00281 V=10.0  +MOVJ EC00281
COMM SMOVC C00282 BC00282 V=10.0  +MOVJ EC00282
COMM SMOVC C00283 BC00283 V=10.0  +MOVJ EC00283
COMM SMOVC C00284 BC00284 V=10.0  +MOVJ EC00284
COMM SMOVC C00285 BC00285 V=10.0  +MOVJ EC00285
COMM ARCOF
COMM SMOVL C00286 BC00286 V=400.0  +MOVJ EC00286
COMM SMOVL C00287 BC00287 V=400.0  +MOVJ EC00287
COMM SFTOF3D
COMM 'Path W1627
COMM SFTOF3D
COMM SFTON3D P022
COMM MOVJ C00288 BC00288 VJ=20.00  +MOVJ EC00288 VJ=100.00
COMM SMOVL C00289 BC00289 V=133.3  +MOVJ EC00289
COMM SMOVL C00290 BC00290 V=100.0 PL=0  +MOVJ EC00290
COMM SREFP 1 C00291 BC00291  +REFP EC00291
COMM SREFP 2 C00292 BC00292  +REFP EC00292
COMM ARCON
COMM SMOVL C00293 BC00293 V=10.0  +MOVJ EC00293
COMM SMOVL C00294 BC00294 V=10.0  +MOVJ EC00294
COMM SMOVL C00295 BC00295 V=13.3  +MOVJ EC00295
COMM ARCOF
COMM SMOVL C00296 BC00296 V=400.0  +MOVJ EC00296
COMM SMOVL C00297 BC00297 V=1000.0  +MOVJ EC00297
COMM SFTOF3D
MOVJ C00298 BC00298 VJ=100.00  +MOVJ EC00298 VJ=100.00
MOVJ C00299 BC00299 VJ=100.00  +MOVJ EC00299 VJ=100.00
MACRO1 MJ#(0) ARGF14
SFTON3D P066
SMOVL C00300 BC00300 V=166.7  +MOVJ EC00300
ARCON
SMOVL C00301 BC00301 V=11.7  +MOVJ EC00301
ARCOF
SMOVL C00302 BC00302 V=333.3  +MOVJ EC00302
SFTOF3D
MOVJ C00303 BC00303 VJ=100.00  +MOVJ EC00303 VJ=100.00
MOVJ C00304 BC00304 VJ=100.00  +MOVJ EC00304 VJ=100.00
SMOVL C00305 BC00305 V=666.7  +MOVJ EC00305
SFTON3D P068
SMOVL C00306 BC00306 V=166.7  +MOVJ EC00306
ARCON
SMOVL C00307 BC00307 V=12.5  +MOVJ EC00307
SMOVL C00308 BC00308 V=10.8  +MOVJ EC00308
SMOVL C00309 BC00309 V=10.8  +MOVJ EC00309
ARCOF
SMOVL C00310 BC00310 V=166.7  +MOVJ EC00310
SMOVL C00311 BC00311 V=666.7  +MOVJ EC00311
SFTOF3D
SMOVL C00312 BC00312 V=666.7  +MOVJ EC00312
'
MOVJ C00313 BC00313 VJ=100.00  +MOVJ EC00313 VJ=100.00
MOVJ C00314 BC00314 VJ=100.00  +MOVJ EC00314 VJ=100.00
MOVJ C00315 BC00315 VJ=100.00  +MOVJ EC00315 VJ=100.00
'Path W1911
SFTOF3D
MOVJ C00316 BC00316 VJ=100.00  +MOVJ EC00316 VJ=100.00
SMOVL C00317 BC00317 V=166.7  +MOVJ EC00317
SFTON3D P021
SMOVL C00318 BC00318 V=100.0 PL=0  +MOVJ EC00318
SREFP 1 C00319 BC00319  +REFP EC00319
SREFP 2 C00320 BC00320  +REFP EC00320
MACRO1 MJ#(0) ARGF21
ARCON
SWVON WEV#(100)
SMOVC C00321 BC00321 V=9.2  +MOVJ EC00321
SMOVC C00322 BC00322 V=9.2  +MOVJ EC00322
SMOVC C00323 BC00323 V=9.2  +MOVJ EC00323
SMOVC C00324 BC00324 V=9.2  +MOVJ EC00324
ARCOF
SWVOF
SMOVL C00325 BC00325 V=400.0  +MOVJ EC00325
SMOVL C00326 BC00326 V=1000.0  +MOVJ EC00326
SFTOF3D
MOVJ C00327 BC00327 VJ=100.00  +MOVJ EC00327 VJ=100.00
'
MOVJ C00328 BC00328 VJ=100.00  +MOVJ EC00328 VJ=100.00
MOVJ C00329 BC00329 VJ=100.00  +MOVJ EC00329 VJ=100.00
'NIE SPAWAMY
COMM 'Path W1642
COMM SFTOF3D
COMM SFTON3D P024
COMM MOVJ C00330 BC00330 VJ=100.00  +MOVJ EC00330 VJ=100.00
COMM SMOVL C00331 BC00331 V=400.0  +MOVJ EC00331
COMM SMOVL C00332 BC00332 V=100.0 PL=0  +MOVJ EC00332
COMM SREFP 1 C00333 BC00333  +REFP EC00333
COMM SREFP 2 C00334 BC00334  +REFP EC00334
COMM MACRO1 MJ#(0) ARGF0
COMM ARCON
COMM SMOVL C00335 BC00335 V=10.0  +MOVJ EC00335
COMM ARCOF
COMM SMOVL C00336 BC00336 V=400.0  +MOVJ EC00336
COMM SMOVL C00337 BC00337 V=1000.0  +MOVJ EC00337
COMM SFTOF3D
'NIE SPAWAMY
COMM 'Path W1643
COMM SFTOF3D
COMM SFTON3D P025
COMM MOVJ C00338 BC00338 VJ=100.00  +MOVJ EC00338 VJ=100.00
COMM SMOVL C00339 BC00339 V=400.0  +MOVJ EC00339
COMM SMOVL C00340 BC00340 V=100.0 PL=0  +MOVJ EC00340
COMM SREFP 1 C00341 BC00341  +REFP EC00341
COMM SREFP 2 C00342 BC00342  +REFP EC00342
COMM MACRO1 MJ#(0) ARGF0
COMM ARCON
COMM SMOVL C00343 BC00343 V=10.0  +MOVJ EC00343
COMM ARCOF
COMM SMOVL C00344 BC00344 V=400.0  +MOVJ EC00344
COMM SMOVL C00345 BC00345 V=1000.0  +MOVJ EC00345
COMM SMOVL C00346 BC00346 V=1000.0  +MOVJ EC00346
COMM SFTOF3D
'
'Path W1644
SFTOF3D
SFTON3D P026
MOVJ C00347 BC00347 VJ=100.00  +MOVJ EC00347 VJ=100.00
SMOVL C00348 BC00348 V=333.3  +MOVJ EC00348
SMOVL C00349 BC00349 V=133.3 PL=0  +MOVJ EC00349
SREFP 1 C00350 BC00350  +REFP EC00350
SREFP 2 C00351 BC00351  +REFP EC00351
MACRO1 MJ#(0) ARGF9
ARCON
SMOVL C00352 BC00352 V=6.7  +MOVJ EC00352
SMOVL C00353 BC00353 V=6.7  +MOVJ EC00353
SMOVL C00354 BC00354 V=6.7  +MOVJ EC00354
SMOVL C00355 BC00355 V=5.0  +MOVJ EC00355
SMOVL C00356 BC00356 V=5.0  +MOVJ EC00356
SMOVL C00357 BC00357 V=5.0  +MOVJ EC00357
ARCOF
SMOVL C00358 BC00358 V=133.3  +MOVJ EC00358
SMOVL C00359 BC00359 V=333.3  +MOVJ EC00359
SMOVL C00360 BC00360 V=333.3  +MOVJ EC00360
SFTOF3D
'Path W1645
SFTOF3D
SFTON3D P027
MOVJ C00361 BC00361 VJ=50.00  +MOVJ EC00361 VJ=100.00
SMOVL C00362 BC00362 V=166.7  +MOVJ EC00362
SMOVL C00363 BC00363 V=133.3 PL=0  +MOVJ EC00363
SREFP 1 C00364 BC00364  +REFP EC00364
SREFP 2 C00365 BC00365  +REFP EC00365
MACRO1 MJ#(0) ARGF9
ARCON
SMOVL C00366 BC00366 V=6.7  +MOVJ EC00366
SMOVL C00367 BC00367 V=6.7  +MOVJ EC00367
SMOVL C00368 BC00368 V=6.7  +MOVJ EC00368
ARCON
SMOVL C00369 BC00369 V=6.7  +MOVJ EC00369
SMOVL C00370 BC00370 V=6.7  +MOVJ EC00370
ARCOF
SMOVL C00371 BC00371 V=400.0  +MOVJ EC00371
SMOVL C00372 BC00372 V=1000.0  +MOVJ EC00372
SMOVL C00373 BC00373 V=1000.0  +MOVJ EC00373
SFTOF3D
MOVJ C00374 BC00374 VJ=40.00  +MOVJ EC00374 VJ=100.00
MOVJ C00375 BC00375 VJ=100.00  +MOVJ EC00375 VJ=100.00
COMM 'jakie searche do takicj spoin?
COMM MOVJ C00376 BC00376 VJ=100.00  +MOVJ EC00376 VJ=100.00
COMM 'Path W1646
COMM SFTOF3D
COMM MOVJ C00377 BC00377 VJ=100.00  +MOVJ EC00377 VJ=100.00
COMM MOVL C00378 BC00378 V=400.0  +MOVJ EC00378 VJ=100.00
COMM PAUSE
COMM PAUSE
'USUNAC SPAWANIE ZAMKOW
COMM SFTOF3D
COMM SFTON3D P021
COMM SMOVL C00379 BC00379 V=166.7 PL=0  +MOVJ EC00379
COMM SREFP 1 C00380 BC00380  +REFP EC00380
COMM SREFP 2 C00381 BC00381  +REFP EC00381
COMM MACRO1 MJ#(0) ARGF6
COMM ARCON
COMM SMOVL C00382 BC00382 V=4.2  +MOVJ EC00382
COMM ARCOF
COMM MOVL C00383 BC00383 V=400.0  +MOVJ EC00383 VJ=100.00
COMM MOVL C00384 BC00384 V=1000.0  +MOVJ EC00384 VJ=100.00
COMM MOVL C00385 BC00385 V=333.3  +MOVJ EC00385 VJ=100.00
COMM MOVJ C00386 BC00386 VJ=100.00  +MOVJ EC00386 VJ=100.00
COMM 'brak dostÄpu do jednej spoiny
COMM 'Path W1647
COMM SFTOF3D
COMM MOVJ C00387 BC00387 VJ=25.00  +MOVJ EC00387 VJ=100.00
COMM MOVJ C00388 BC00388 VJ=25.00  +MOVJ EC00388 VJ=100.00
COMM MOVL C00389 BC00389 V=400.0  +MOVJ EC00389 VJ=100.00
COMM SFTOF3D
COMM SMOVL C00390 BC00390 V=166.7 PL=0  +MOVJ EC00390
COMM SREFP 1 C00391 BC00391  +REFP EC00391
COMM SREFP 2 C00392 BC00392  +REFP EC00392
COMM MACRO1 MJ#(0) ARGF6
COMM ARCON
COMM SMOVL C00393 BC00393 V=4.2  +MOVJ EC00393
COMM ARCOF
COMM MOVL C00394 BC00394 V=400.0  +MOVJ EC00394 VJ=100.00
COMM MOVL C00395 BC00395 V=1000.0  +MOVJ EC00395 VJ=100.00
COMM 'Path W1648
COMM SFTOF3D
COMM MOVJ C00396 BC00396 VJ=10.00  +MOVJ EC00396 VJ=100.00
COMM MOVL C00397 BC00397 V=166.7  +MOVJ EC00397 VJ=100.00
COMM SFTON3D P021
COMM SMOVL C00398 BC00398 V=100.0 PL=0  +MOVJ EC00398
COMM SREFP 1 C00399 BC00399  +REFP EC00399
COMM SREFP 2 C00400 BC00400  +REFP EC00400
COMM MACRO1 MJ#(0) ARGF6
COMM ARCON
COMM SMOVL C00401 BC00401 V=4.2  +MOVJ EC00401
COMM ARCOF
COMM MOVL C00402 BC00402 V=400.0  +MOVJ EC00402 VJ=100.00
COMM MOVL C00403 BC00403 V=1000.0  +MOVJ EC00403 VJ=100.00
COMM MOVL C00404 BC00404 V=1000.0  +MOVJ EC00404 VJ=100.00
COMM MOVJ C00405 BC00405 VJ=10.00  +MOVJ EC00405 VJ=100.00
COMM 'Path W1649
COMM SFTOF3D
COMM MOVJ C00406 BC00406 VJ=15.00  +MOVJ EC00406 VJ=100.00
COMM MOVL C00407 BC00407 V=166.7  +MOVJ EC00407 VJ=100.00
COMM SFTON3D P021
COMM SMOVL C00408 BC00408 V=166.7 PL=0  +MOVJ EC00408
COMM SREFP 1 C00409 BC00409  +REFP EC00409
COMM SREFP 2 C00410 BC00410  +REFP EC00410
COMM MACRO1 MJ#(0) ARGF6
COMM ARCON
COMM SMOVL C00411 BC00411 V=4.2  +MOVJ EC00411
COMM ARCOF
COMM MOVL C00412 BC00412 V=400.0  +MOVJ EC00412 VJ=100.00
COMM MOVL C00413 BC00413 V=1000.0  +MOVJ EC00413 VJ=100.00
COMM 'Path W1650
COMM MOVJ C00414 BC00414 VJ=100.00  +MOVJ EC00414 VJ=100.00
COMM MOVL C00415 BC00415 V=166.7  +MOVJ EC00415 VJ=100.00
COMM SMOVL C00416 BC00416 V=166.7 PL=0  +MOVJ EC00416
COMM SREFP 1 C00417 BC00417  +REFP EC00417
COMM SREFP 2 C00418 BC00418  +REFP EC00418
COMM MACRO1 MJ#(0) ARGF6
COMM ARCON
COMM SMOVL C00419 BC00419 V=4.2  +MOVJ EC00419
COMM ARCOF
COMM MOVL C00420 BC00420 V=400.0  +MOVJ EC00420 VJ=100.00
COMM MOVL C00421 BC00421 V=1000.0  +MOVJ EC00421 VJ=100.00
COMM 'Path W1651
COMM SFTOF3D
COMM MOVJ C00422 BC00422 VJ=100.00  +MOVJ EC00422 VJ=100.00
COMM MOVL C00423 BC00423 V=400.0  +MOVJ EC00423 VJ=100.00
COMM SFTON3D P021
COMM SMOVL C00424 BC00424 V=166.7 PL=0  +MOVJ EC00424
COMM SREFP 1 C00425 BC00425  +REFP EC00425
COMM SREFP 2 C00426 BC00426  +REFP EC00426
COMM MACRO1 MJ#(0) ARGF6
COMM ARCON
COMM SMOVL C00427 BC00427 V=4.2  +MOVJ EC00427
COMM ARCOF
COMM MOVL C00428 BC00428 V=400.0  +MOVJ EC00428 VJ=100.00
COMM MOVL C00429 BC00429 V=1000.0  +MOVJ EC00429 VJ=100.00
COMM 'Path W1652
COMM SFTOF3D
COMM MOVJ C00430 BC00430 VJ=100.00  +MOVJ EC00430 VJ=100.00
COMM MOVL C00431 BC00431 V=166.7  +MOVJ EC00431 VJ=100.00
COMM SFTON3D P021
COMM SMOVL C00432 BC00432 V=166.7 PL=0  +MOVJ EC00432
COMM SREFP 1 C00433 BC00433  +REFP EC00433
COMM SREFP 2 C00434 BC00434  +REFP EC00434
COMM MACRO1 MJ#(0) ARGF6
COMM ARCON
COMM SMOVL C00435 BC00435 V=4.2  +MOVJ EC00435
COMM ARCOF
COMM MOVL C00436 BC00436 V=166.7  +MOVJ EC00436 VJ=100.00
COMM MOVL C00437 BC00437 V=166.7  +MOVJ EC00437 VJ=100.00
COMM MOVJ C00438 BC00438 VJ=50.00  +MOVJ EC00438 VJ=20.00
COMM SMOVL C00439 BC00439 V=166.7  +MOVJ EC00439
COMM ARCON
COMM SMOVL C00440 BC00440 V=4.2  +MOVJ EC00440
COMM ARCOF
COMM SMOVL C00441 BC00441 V=166.7  +MOVJ EC00441
COMM 'jakie searche do takicj spoin?
COMM MOVJ C00442 BC00442 VJ=100.00  +MOVJ EC00442 VJ=100.00
COMM MOVJ C00443 BC00443 VJ=20.00  +MOVJ EC00443 VJ=100.00
COMM MOVJ C00444 BC00444 VJ=100.00  +MOVJ EC00444 VJ=100.00
COMM MOVJ C00445 BC00445 VJ=100.00  +MOVJ EC00445 VJ=100.00
COMM 'Path W1653
COMM SFTOF3D
COMM MOVJ C00446 BC00446 VJ=100.00  +MOVJ EC00446 VJ=100.00
COMM MOVL C00447 BC00447 V=166.7  +MOVJ EC00447 VJ=100.00
COMM SFTON3D P067
COMM SMOVL C00448 BC00448 V=166.7 PL=0  +MOVJ EC00448
COMM SREFP 1 C00449 BC00449  +REFP EC00449
COMM SREFP 2 C00450 BC00450  +REFP EC00450
COMM ARCON
COMM MACRO1 MJ#(0) ARGF9
COMM SMOVL C00451 BC00451 V=10.8  +MOVJ EC00451
COMM ARCOF
COMM SMOVL C00452 BC00452 V=166.7  +MOVJ EC00452
COMM SMOVL C00453 BC00453 V=666.7  +MOVJ EC00453
COMM SMOVL C00454 BC00454 V=166.7  +MOVJ EC00454
COMM ARCON
COMM SMOVL C00455 BC00455 V=10.8  +MOVJ EC00455
COMM ARCOF
COMM SMOVL C00456 BC00456 V=250.0  +MOVJ EC00456
COMM 'Path W1654
COMM SFTOF3D
COMM MOVJ C00457 BC00457 VJ=100.00  +MOVJ EC00457 VJ=100.00
COMM MOVJ C00458 BC00458 VJ=100.00  +MOVJ EC00458 VJ=100.00
MOVJ C00459 BC00459 VJ=100.00  +MOVJ EC00459 VJ=100.00
'Down
END
